REGION Network 6: InterLock
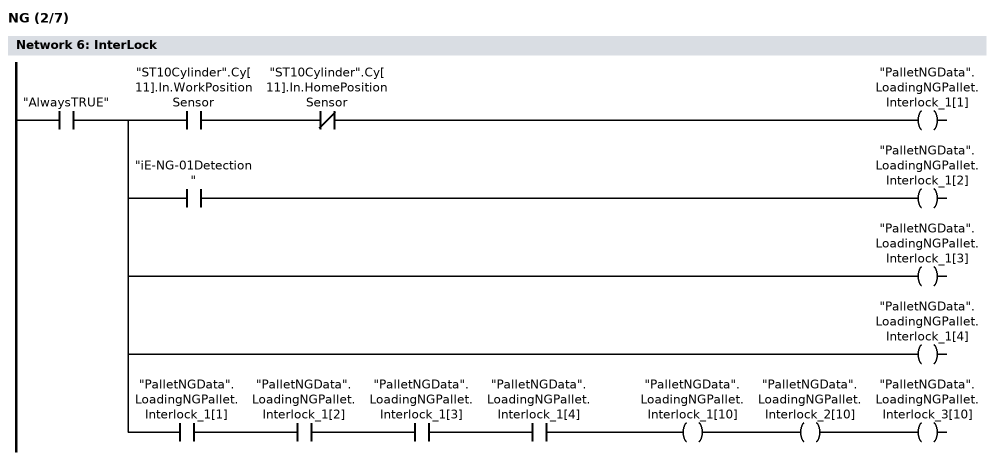
   RUNG wire#powerrail
      Contact( "AlwaysTRUE" )
      wire#w1
      Contact( "ST10Cylinder".Cy[11].In.WorkPositionSensor )
      I_Contact( "ST10Cylinder".Cy[11].In.HomePositionSensor )
      Coil( "PalletNGData".LoadingNGPallet.Interlock_1[1] )
   END_RUNG
   RUNG wire#w1
      Contact( "iE-NG-01Detection" )
      Coil( "PalletNGData".LoadingNGPallet.Interlock_1[2] )
   END_RUNG
   RUNG wire#w1
      Coil( "PalletNGData".LoadingNGPallet.Interlock_1[3] )
   END_RUNG
   RUNG wire#w1
      Coil( "PalletNGData".LoadingNGPallet.Interlock_1[4] )
   END_RUNG
   RUNG wire#w1
      Contact( "PalletNGData".LoadingNGPallet.Interlock_1[1] )
      Contact( "PalletNGData".LoadingNGPallet.Interlock_1[2] )
      Contact( "PalletNGData".LoadingNGPallet.Interlock_1[3] )
      Contact( "PalletNGData".LoadingNGPallet.Interlock_1[4] )
      Coil( "PalletNGData".LoadingNGPallet.Interlock_1[10] )
      Coil( "PalletNGData".LoadingNGPallet.Interlock_2[10] )
      Coil( "PalletNGData".LoadingNGPallet.Interlock_3[10] )
   END_RUNG
   // the same network as SCL:
   "PalletNGData".LoadingNGPallet.Interlock_1[1] := "AlwaysTRUE" AND "ST10Cylinder".Cy[11].In.WorkPositionSensor AND NOT "ST10Cylinder".Cy[11].In.HomePositionSensor;
   "PalletNGData".LoadingNGPallet.Interlock_1[2] := "AlwaysTRUE" AND "iE-NG-01Detection";
   "PalletNGData".LoadingNGPallet.Interlock_1[3] := "AlwaysTRUE";
   "PalletNGData".LoadingNGPallet.Interlock_1[4] := "AlwaysTRUE";
   #_w1 := "AlwaysTRUE" AND "PalletNGData".LoadingNGPallet.Interlock_1[1] AND "PalletNGData".LoadingNGPallet.Interlock_1[2] AND "PalletNGData".LoadingNGPallet.Interlock_1[3] AND "PalletNGData".LoadingNGPallet.Interlock_1[4];
   "PalletNGData".LoadingNGPallet.Interlock_1[10] := #_w1;
   "PalletNGData".LoadingNGPallet.Interlock_2[10] := #_w1;
   "PalletNGData".LoadingNGPallet.Interlock_3[10] := #_w1;
END_REGION

REGION Network 7: NG_Button
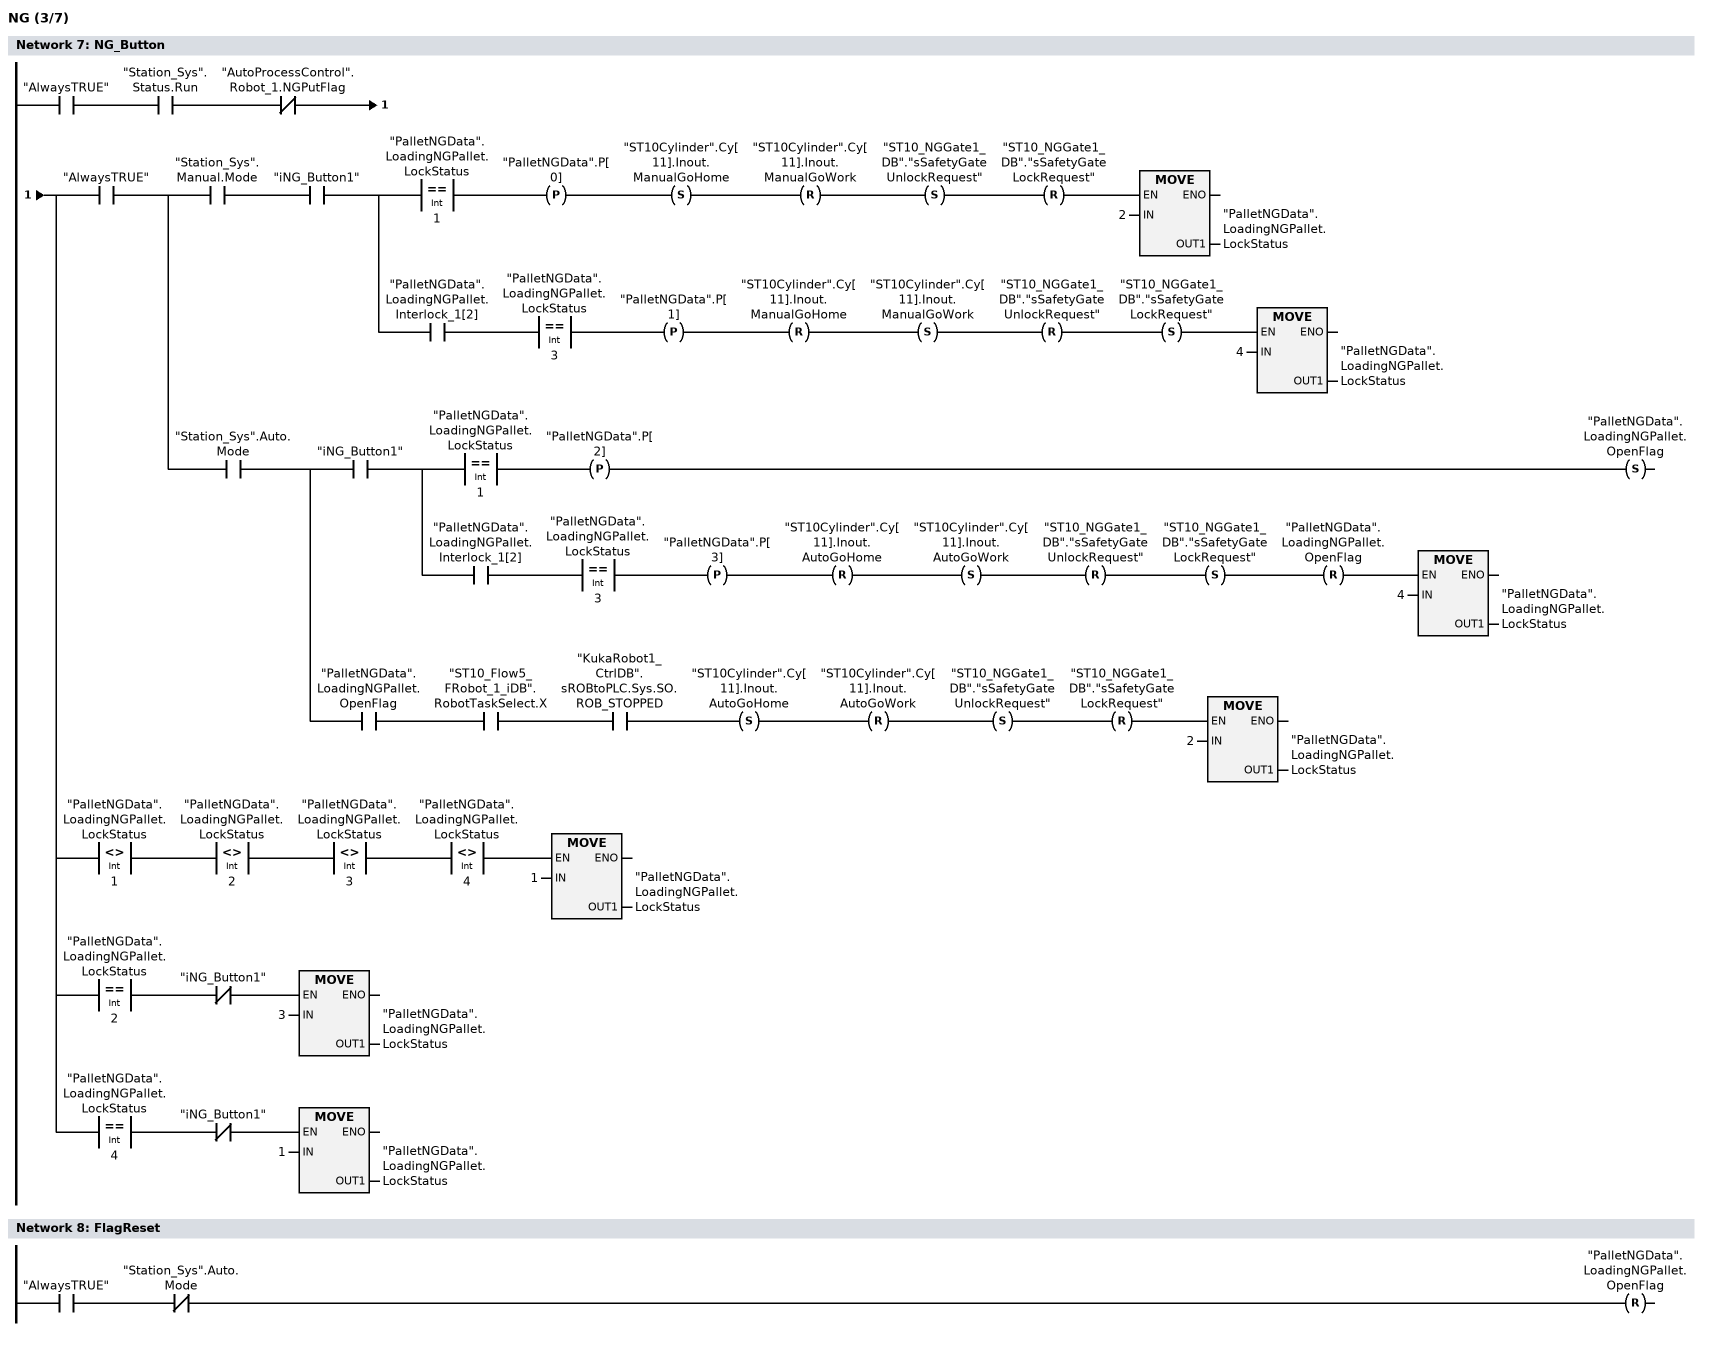
   RUNG wire#powerrail
      Contact( "AlwaysTRUE" )
      Contact( "Station_Sys".Status.Run )
      I_Contact( "AutoProcessControl".Robot_1.NGPutFlag )
      wire#w1
      Contact( "AlwaysTRUE" )
      wire#w2
      Contact( "Station_Sys".Manual.Mode )
      Contact( "iNG_Button1" )
      wire#w3
      { S7_Templates := "SrcType := Int" } EQ_Contact(in1 := "PalletNGData".LoadingNGPallet.LockStatus, in2 := 1)
      P_Trig( "PalletNGData".P[0] )
      S_Coil( "ST10Cylinder".Cy[11].Inout.ManualGoHome )
      R_Coil( "ST10Cylinder".Cy[11].Inout.ManualGoWork )
      S_Coil( "ST10_NGGate1_DB"."sSafetyGate UnlockRequest" )
      R_Coil( "ST10_NGGate1_DB"."sSafetyGate LockRequest" )
      Move(in := 2, out1 => "PalletNGData".LoadingNGPallet.LockStatus)
   END_RUNG
   RUNG wire#w3
      Contact( "PalletNGData".LoadingNGPallet.Interlock_1[2] )
      { S7_Templates := "SrcType := Int" } EQ_Contact(in1 := "PalletNGData".LoadingNGPallet.LockStatus, in2 := 3)
      P_Trig( "PalletNGData".P[1] )
      R_Coil( "ST10Cylinder".Cy[11].Inout.ManualGoHome )
      S_Coil( "ST10Cylinder".Cy[11].Inout.ManualGoWork )
      R_Coil( "ST10_NGGate1_DB"."sSafetyGate UnlockRequest" )
      S_Coil( "ST10_NGGate1_DB"."sSafetyGate LockRequest" )
      Move(in := 4, out1 => "PalletNGData".LoadingNGPallet.LockStatus)
   END_RUNG
   RUNG wire#w2
      Contact( "Station_Sys".Auto.Mode )
      wire#w4
      Contact( "iNG_Button1" )
      wire#w5
      { S7_Templates := "SrcType := Int" } EQ_Contact(in1 := "PalletNGData".LoadingNGPallet.LockStatus, in2 := 1)
      P_Trig( "PalletNGData".P[2] )
      S_Coil( "PalletNGData".LoadingNGPallet.OpenFlag )
   END_RUNG
   RUNG wire#w5
      Contact( "PalletNGData".LoadingNGPallet.Interlock_1[2] )
      { S7_Templates := "SrcType := Int" } EQ_Contact(in1 := "PalletNGData".LoadingNGPallet.LockStatus, in2 := 3)
      P_Trig( "PalletNGData".P[3] )
      R_Coil( "ST10Cylinder".Cy[11].Inout.AutoGoHome )
      S_Coil( "ST10Cylinder".Cy[11].Inout.AutoGoWork )
      R_Coil( "ST10_NGGate1_DB"."sSafetyGate UnlockRequest" )
      S_Coil( "ST10_NGGate1_DB"."sSafetyGate LockRequest" )
      R_Coil( "PalletNGData".LoadingNGPallet.OpenFlag )
      Move(in := 4, out1 => "PalletNGData".LoadingNGPallet.LockStatus)
   END_RUNG
   RUNG wire#w4
      Contact( "PalletNGData".LoadingNGPallet.OpenFlag )
      Contact( "ST10_Flow5_FRobot_1_iDB".RobotTaskSelect.X )
      Contact( "KukaRobot1_CtrlDB".sROBtoPLC.Sys.SO.ROB_STOPPED )
      S_Coil( "ST10Cylinder".Cy[11].Inout.AutoGoHome )
      R_Coil( "ST10Cylinder".Cy[11].Inout.AutoGoWork )
      S_Coil( "ST10_NGGate1_DB"."sSafetyGate UnlockRequest" )
      R_Coil( "ST10_NGGate1_DB"."sSafetyGate LockRequest" )
      Move(in := 2, out1 => "PalletNGData".LoadingNGPallet.LockStatus)
   END_RUNG
   RUNG wire#w1
      { S7_Templates := "SrcType := Int" } NE_Contact(in1 := "PalletNGData".LoadingNGPallet.LockStatus, in2 := 1)
      { S7_Templates := "SrcType := Int" } NE_Contact(in1 := "PalletNGData".LoadingNGPallet.LockStatus, in2 := 2)
      { S7_Templates := "SrcType := Int" } NE_Contact(in1 := "PalletNGData".LoadingNGPallet.LockStatus, in2 := 3)
      { S7_Templates := "SrcType := Int" } NE_Contact(in1 := "PalletNGData".LoadingNGPallet.LockStatus, in2 := 4)
      Move(in := 1, out1 => "PalletNGData".LoadingNGPallet.LockStatus)
   END_RUNG
   RUNG wire#w1
      { S7_Templates := "SrcType := Int" } EQ_Contact(in1 := "PalletNGData".LoadingNGPallet.LockStatus, in2 := 2)
      I_Contact( "iNG_Button1" )
      Move(in := 3, out1 => "PalletNGData".LoadingNGPallet.LockStatus)
   END_RUNG
   RUNG wire#w1
      { S7_Templates := "SrcType := Int" } EQ_Contact(in1 := "PalletNGData".LoadingNGPallet.LockStatus, in2 := 4)
      I_Contact( "iNG_Button1" )
      Move(in := 1, out1 => "PalletNGData".LoadingNGPallet.LockStatus)
   END_RUNG
   // the same network as SCL:
   #_w1 := "AlwaysTRUE" AND "Station_Sys".Status.Run AND NOT "AutoProcessControl".Robot_1.NGPutFlag;
   #_w2 := #_w1 AND "AlwaysTRUE";
   #_w3 := #_w2 AND "Station_Sys".Manual.Mode AND "iNG_Button1";
   #_w4 := #_w3 AND ("PalletNGData".LoadingNGPallet.LockStatus = 1);
   #_w5 := #_w4 AND NOT "PalletNGData".P[0];   // rising edge
   "PalletNGData".P[0] := #_w4;
   IF #_w5 THEN
       "ST10Cylinder".Cy[11].Inout.ManualGoHome := TRUE;
       "ST10Cylinder".Cy[11].Inout.ManualGoWork := FALSE;
       "ST10_NGGate1_DB"."sSafetyGate UnlockRequest" := TRUE;
       "ST10_NGGate1_DB"."sSafetyGate LockRequest" := FALSE;
       "PalletNGData".LoadingNGPallet.LockStatus := 2;
   END_IF;
   #_w6 := #_w3 AND "PalletNGData".LoadingNGPallet.Interlock_1[2] AND ("PalletNGData".LoadingNGPallet.LockStatus = 3);
   #_w7 := #_w6 AND NOT "PalletNGData".P[1];   // rising edge
   "PalletNGData".P[1] := #_w6;
   IF #_w7 THEN
       "ST10Cylinder".Cy[11].Inout.ManualGoHome := FALSE;
       "ST10Cylinder".Cy[11].Inout.ManualGoWork := TRUE;
       "ST10_NGGate1_DB"."sSafetyGate UnlockRequest" := FALSE;
       "ST10_NGGate1_DB"."sSafetyGate LockRequest" := TRUE;
       "PalletNGData".LoadingNGPallet.LockStatus := 4;
   END_IF;
   #_w8 := #_w2 AND "Station_Sys".Auto.Mode;
   #_w9 := #_w8 AND "iNG_Button1";
   #_w10 := #_w9 AND ("PalletNGData".LoadingNGPallet.LockStatus = 1);
   #_w11 := #_w10 AND NOT "PalletNGData".P[2];   // rising edge
   "PalletNGData".P[2] := #_w10;
   IF #_w11 THEN "PalletNGData".LoadingNGPallet.OpenFlag := TRUE; END_IF;
   #_w12 := #_w9 AND "PalletNGData".LoadingNGPallet.Interlock_1[2] AND ("PalletNGData".LoadingNGPallet.LockStatus = 3);
   #_w13 := #_w12 AND NOT "PalletNGData".P[3];   // rising edge
   "PalletNGData".P[3] := #_w12;
   IF #_w13 THEN
       "ST10Cylinder".Cy[11].Inout.AutoGoHome := FALSE;
       "ST10Cylinder".Cy[11].Inout.AutoGoWork := TRUE;
       "ST10_NGGate1_DB"."sSafetyGate UnlockRequest" := FALSE;
       "ST10_NGGate1_DB"."sSafetyGate LockRequest" := TRUE;
       "PalletNGData".LoadingNGPallet.OpenFlag := FALSE;
       "PalletNGData".LoadingNGPallet.LockStatus := 4;
   END_IF;
   IF #_w8 AND "PalletNGData".LoadingNGPallet.OpenFlag AND "ST10_Flow5_FRobot_1_iDB".RobotTaskSelect.X AND "KukaRobot1_CtrlDB".sROBtoPLC.Sys.SO.ROB_STOPPED THEN
       "ST10Cylinder".Cy[11].Inout.AutoGoHome := TRUE;
       "ST10Cylinder".Cy[11].Inout.AutoGoWork := FALSE;
       "ST10_NGGate1_DB"."sSafetyGate UnlockRequest" := TRUE;
       "ST10_NGGate1_DB"."sSafetyGate LockRequest" := FALSE;
       "PalletNGData".LoadingNGPallet.LockStatus := 2;
   END_IF;
   IF #_w1 AND ("PalletNGData".LoadingNGPallet.LockStatus <> 1) AND ("PalletNGData".LoadingNGPallet.LockStatus <> 2) AND ("PalletNGData".LoadingNGPallet.LockStatus <> 3) AND ("PalletNGData".LoadingNGPallet.LockStatus <> 4) THEN
       "PalletNGData".LoadingNGPallet.LockStatus := 1;
   END_IF;
   IF #_w1 AND ("PalletNGData".LoadingNGPallet.LockStatus = 2) AND NOT "iNG_Button1" THEN
       "PalletNGData".LoadingNGPallet.LockStatus := 3;
   END_IF;
   IF #_w1 AND ("PalletNGData".LoadingNGPallet.LockStatus = 4) AND NOT "iNG_Button1" THEN
       "PalletNGData".LoadingNGPallet.LockStatus := 1;
   END_IF;
END_REGION

REGION Network 8: FlagReset
   RUNG wire#powerrail
      Contact( "AlwaysTRUE" )
      I_Contact( "Station_Sys".Auto.Mode )
      R_Coil( "PalletNGData".LoadingNGPallet.OpenFlag )
   END_RUNG
   // the same network as SCL:
   IF "AlwaysTRUE" AND NOT "Station_Sys".Auto.Mode THEN
       "PalletNGData".LoadingNGPallet.OpenFlag := FALSE;
   END_IF;
END_REGION

REGION Network 9: NG Door
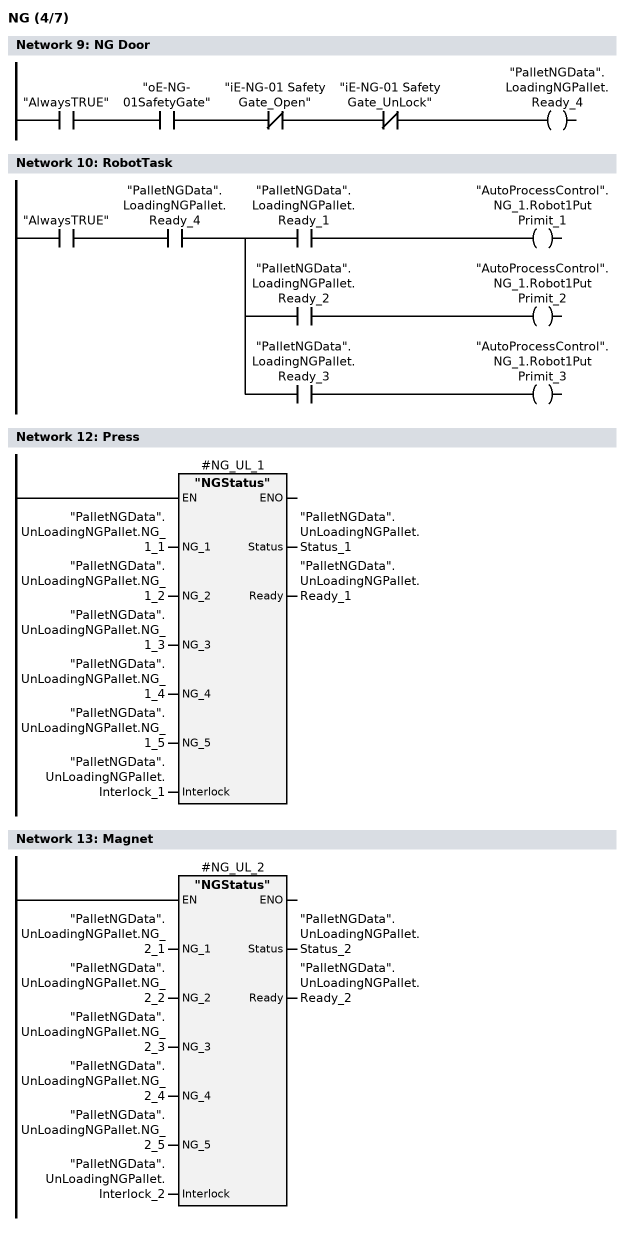
   RUNG wire#powerrail
      Contact( "AlwaysTRUE" )
      Contact( "oE-NG-01SafetyGate" )
      I_Contact( "iE-NG-01 Safety Gate_Open" )
      I_Contact( "iE-NG-01 Safety Gate_UnLock" )
      Coil( "PalletNGData".LoadingNGPallet.Ready_4 )
   END_RUNG
   // the same network as SCL:
   "PalletNGData".LoadingNGPallet.Ready_4 := "AlwaysTRUE" AND "oE-NG-01SafetyGate" AND NOT "iE-NG-01 Safety Gate_Open" AND NOT "iE-NG-01 Safety Gate_UnLock";
END_REGION

REGION Network 10: RobotTask
   RUNG wire#powerrail
      Contact( "AlwaysTRUE" )
      Contact( "PalletNGData".LoadingNGPallet.Ready_4 )
      wire#w1
      Contact( "PalletNGData".LoadingNGPallet.Ready_1 )
      Coil( "AutoProcessControl".NG_1.Robot1PutPrimit_1 )
   END_RUNG
   RUNG wire#w1
      Contact( "PalletNGData".LoadingNGPallet.Ready_2 )
      Coil( "AutoProcessControl".NG_1.Robot1PutPrimit_2 )
   END_RUNG
   RUNG wire#w1
      Contact( "PalletNGData".LoadingNGPallet.Ready_3 )
      Coil( "AutoProcessControl".NG_1.Robot1PutPrimit_3 )
   END_RUNG
   // the same network as SCL:
   #_w1 := "AlwaysTRUE" AND "PalletNGData".LoadingNGPallet.Ready_4;
   "AutoProcessControl".NG_1.Robot1PutPrimit_1 := #_w1 AND "PalletNGData".LoadingNGPallet.Ready_1;
   "AutoProcessControl".NG_1.Robot1PutPrimit_2 := #_w1 AND "PalletNGData".LoadingNGPallet.Ready_2;
   "AutoProcessControl".NG_1.Robot1PutPrimit_3 := #_w1 AND "PalletNGData".LoadingNGPallet.Ready_3;
END_REGION

REGION Network 11: --------------------------------------- UnLoad -------------------------------------------------------
END_REGION

REGION Network 12: Press
   RUNG wire#powerrail
      #NG_UL_1(NG_1 := "PalletNGData".UnLoadingNGPallet.NG_1_1, NG_2 := "PalletNGData".UnLoadingNGPallet.NG_1_2, NG_3 := "PalletNGData".UnLoadingNGPallet.NG_1_3, NG_4 := "PalletNGData".UnLoadingNGPallet.NG_1_4, NG_5 := "PalletNGData".UnLoadingNGPallet.NG_1_5, Interlock := "PalletNGData".UnLoadingNGPallet.Interlock_1, Status => "PalletNGData".UnLoadingNGPallet.Status_1, Ready => "PalletNGData".UnLoadingNGPallet.Ready_1)
   END_RUNG
   // the same network as SCL:
   #NG_UL_1(NG_1 := "PalletNGData".UnLoadingNGPallet.NG_1_1,   // "NGStatus"
            NG_2 := "PalletNGData".UnLoadingNGPallet.NG_1_2,
            NG_3 := "PalletNGData".UnLoadingNGPallet.NG_1_3,
            NG_4 := "PalletNGData".UnLoadingNGPallet.NG_1_4,
            NG_5 := "PalletNGData".UnLoadingNGPallet.NG_1_5,
            Interlock := "PalletNGData".UnLoadingNGPallet.Interlock_1,
            Status => "PalletNGData".UnLoadingNGPallet.Status_1,
            Ready => "PalletNGData".UnLoadingNGPallet.Ready_1);
END_REGION

REGION Network 13: Magnet
   RUNG wire#powerrail
      #NG_UL_2(NG_1 := "PalletNGData".UnLoadingNGPallet.NG_2_1, NG_2 := "PalletNGData".UnLoadingNGPallet.NG_2_2, NG_3 := "PalletNGData".UnLoadingNGPallet.NG_2_3, NG_4 := "PalletNGData".UnLoadingNGPallet.NG_2_4, NG_5 := "PalletNGData".UnLoadingNGPallet.NG_2_5, Interlock := "PalletNGData".UnLoadingNGPallet.Interlock_2, Status => "PalletNGData".UnLoadingNGPallet.Status_2, Ready => "PalletNGData".UnLoadingNGPallet.Ready_2)
   END_RUNG
   // the same network as SCL:
   #NG_UL_2(NG_1 := "PalletNGData".UnLoadingNGPallet.NG_2_1,   // "NGStatus"
            NG_2 := "PalletNGData".UnLoadingNGPallet.NG_2_2,
            NG_3 := "PalletNGData".UnLoadingNGPallet.NG_2_3,
            NG_4 := "PalletNGData".UnLoadingNGPallet.NG_2_4,
            NG_5 := "PalletNGData".UnLoadingNGPallet.NG_2_5,
            Interlock := "PalletNGData".UnLoadingNGPallet.Interlock_2,
            Status => "PalletNGData".UnLoadingNGPallet.Status_2,
            Ready => "PalletNGData".UnLoadingNGPallet.Ready_2);
END_REGION

REGION Network 14: Ring
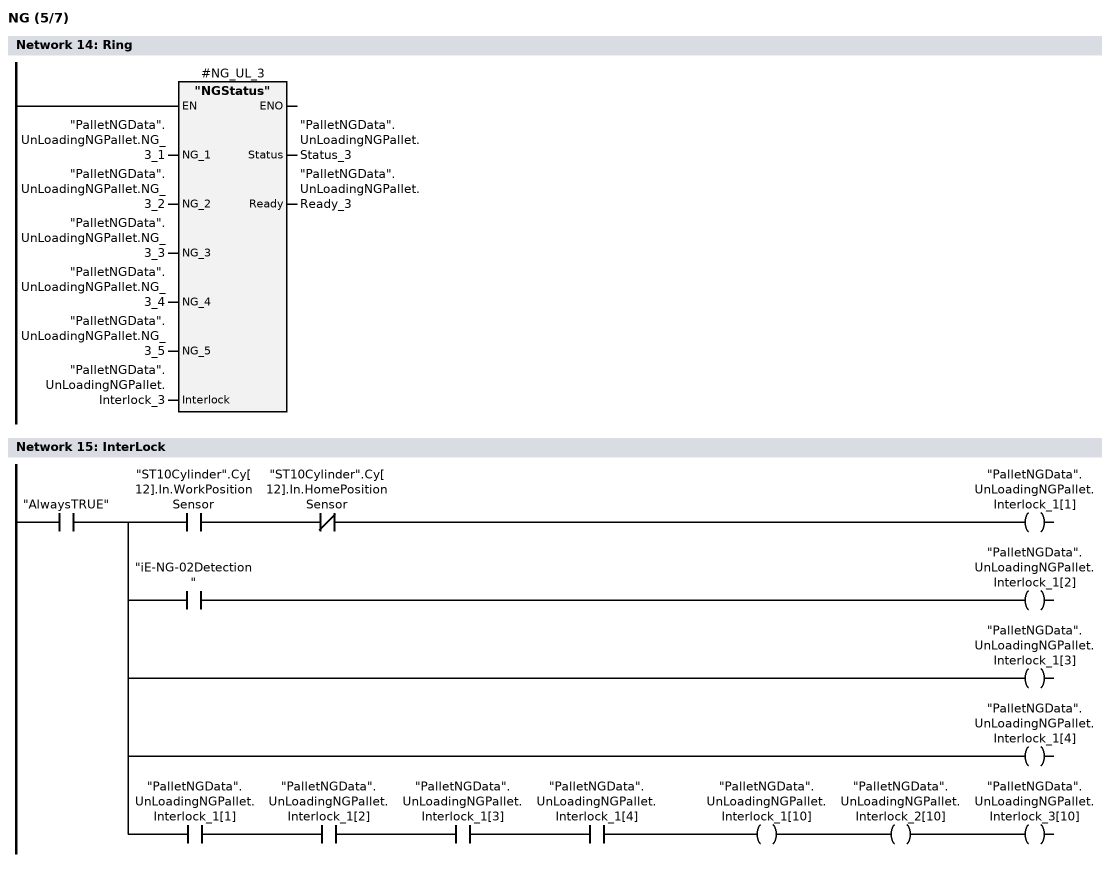
   RUNG wire#powerrail
      #NG_UL_3(NG_1 := "PalletNGData".UnLoadingNGPallet.NG_3_1, NG_2 := "PalletNGData".UnLoadingNGPallet.NG_3_2, NG_3 := "PalletNGData".UnLoadingNGPallet.NG_3_3, NG_4 := "PalletNGData".UnLoadingNGPallet.NG_3_4, NG_5 := "PalletNGData".UnLoadingNGPallet.NG_3_5, Interlock := "PalletNGData".UnLoadingNGPallet.Interlock_3, Status => "PalletNGData".UnLoadingNGPallet.Status_3, Ready => "PalletNGData".UnLoadingNGPallet.Ready_3)
   END_RUNG
   // the same network as SCL:
   #NG_UL_3(NG_1 := "PalletNGData".UnLoadingNGPallet.NG_3_1,   // "NGStatus"
            NG_2 := "PalletNGData".UnLoadingNGPallet.NG_3_2,
            NG_3 := "PalletNGData".UnLoadingNGPallet.NG_3_3,
            NG_4 := "PalletNGData".UnLoadingNGPallet.NG_3_4,
            NG_5 := "PalletNGData".UnLoadingNGPallet.NG_3_5,
            Interlock := "PalletNGData".UnLoadingNGPallet.Interlock_3,
            Status => "PalletNGData".UnLoadingNGPallet.Status_3,
            Ready => "PalletNGData".UnLoadingNGPallet.Ready_3);
END_REGION

REGION Network 15: InterLock
   RUNG wire#powerrail
      Contact( "AlwaysTRUE" )
      wire#w1
      Contact( "ST10Cylinder".Cy[12].In.WorkPositionSensor )
      I_Contact( "ST10Cylinder".Cy[12].In.HomePositionSensor )
      Coil( "PalletNGData".UnLoadingNGPallet.Interlock_1[1] )
   END_RUNG
   RUNG wire#w1
      Contact( "iE-NG-02Detection" )
      Coil( "PalletNGData".UnLoadingNGPallet.Interlock_1[2] )
   END_RUNG
   RUNG wire#w1
      Coil( "PalletNGData".UnLoadingNGPallet.Interlock_1[3] )
   END_RUNG
   RUNG wire#w1
      Coil( "PalletNGData".UnLoadingNGPallet.Interlock_1[4] )
   END_RUNG
   RUNG wire#w1
      Contact( "PalletNGData".UnLoadingNGPallet.Interlock_1[1] )
      Contact( "PalletNGData".UnLoadingNGPallet.Interlock_1[2] )
      Contact( "PalletNGData".UnLoadingNGPallet.Interlock_1[3] )
      Contact( "PalletNGData".UnLoadingNGPallet.Interlock_1[4] )
      Coil( "PalletNGData".UnLoadingNGPallet.Interlock_1[10] )
      Coil( "PalletNGData".UnLoadingNGPallet.Interlock_2[10] )
      Coil( "PalletNGData".UnLoadingNGPallet.Interlock_3[10] )
   END_RUNG
   // the same network as SCL:
   "PalletNGData".UnLoadingNGPallet.Interlock_1[1] := "AlwaysTRUE" AND "ST10Cylinder".Cy[12].In.WorkPositionSensor AND NOT "ST10Cylinder".Cy[12].In.HomePositionSensor;
   "PalletNGData".UnLoadingNGPallet.Interlock_1[2] := "AlwaysTRUE" AND "iE-NG-02Detection";
   "PalletNGData".UnLoadingNGPallet.Interlock_1[3] := "AlwaysTRUE";
   "PalletNGData".UnLoadingNGPallet.Interlock_1[4] := "AlwaysTRUE";
   #_w1 := "AlwaysTRUE" AND "PalletNGData".UnLoadingNGPallet.Interlock_1[1] AND "PalletNGData".UnLoadingNGPallet.Interlock_1[2] AND "PalletNGData".UnLoadingNGPallet.Interlock_1[3] AND "PalletNGData".UnLoadingNGPallet.Interlock_1[4];
   "PalletNGData".UnLoadingNGPallet.Interlock_1[10] := #_w1;
   "PalletNGData".UnLoadingNGPallet.Interlock_2[10] := #_w1;
   "PalletNGData".UnLoadingNGPallet.Interlock_3[10] := #_w1;
END_REGION

REGION Network 16: NG_Button
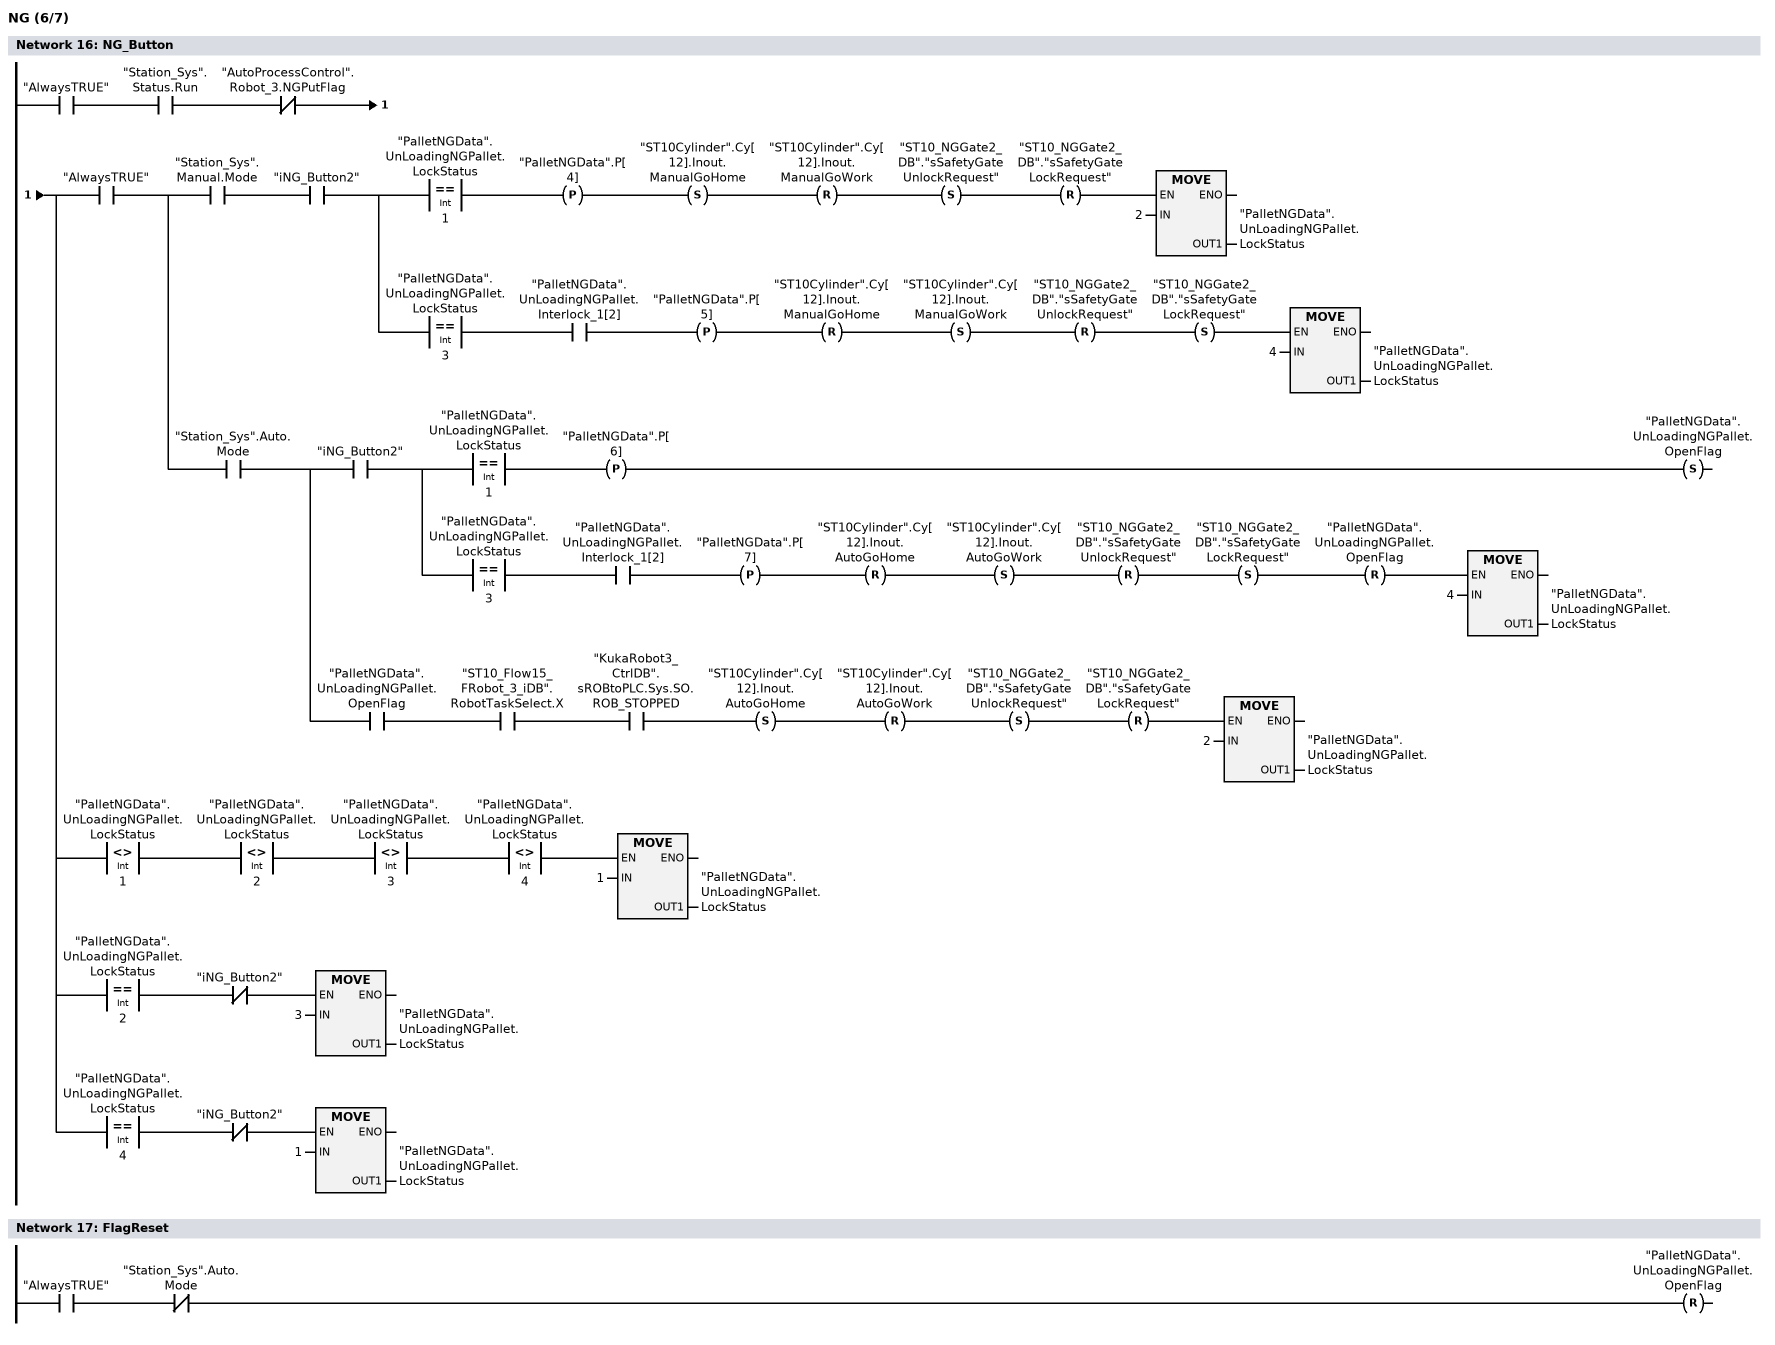
   RUNG wire#powerrail
      Contact( "AlwaysTRUE" )
      Contact( "Station_Sys".Status.Run )
      I_Contact( "AutoProcessControl".Robot_3.NGPutFlag )
      wire#w1
      Contact( "AlwaysTRUE" )
      wire#w2
      Contact( "Station_Sys".Manual.Mode )
      Contact( "iNG_Button2" )
      wire#w3
      { S7_Templates := "SrcType := Int" } EQ_Contact(in1 := "PalletNGData".UnLoadingNGPallet.LockStatus, in2 := 1)
      P_Trig( "PalletNGData".P[4] )
      S_Coil( "ST10Cylinder".Cy[12].Inout.ManualGoHome )
      R_Coil( "ST10Cylinder".Cy[12].Inout.ManualGoWork )
      S_Coil( "ST10_NGGate2_DB"."sSafetyGate UnlockRequest" )
      R_Coil( "ST10_NGGate2_DB"."sSafetyGate LockRequest" )
      Move(in := 2, out1 => "PalletNGData".UnLoadingNGPallet.LockStatus)
   END_RUNG
   RUNG wire#w3
      { S7_Templates := "SrcType := Int" } EQ_Contact(in1 := "PalletNGData".UnLoadingNGPallet.LockStatus, in2 := 3)
      Contact( "PalletNGData".UnLoadingNGPallet.Interlock_1[2] )
      P_Trig( "PalletNGData".P[5] )
      R_Coil( "ST10Cylinder".Cy[12].Inout.ManualGoHome )
      S_Coil( "ST10Cylinder".Cy[12].Inout.ManualGoWork )
      R_Coil( "ST10_NGGate2_DB"."sSafetyGate UnlockRequest" )
      S_Coil( "ST10_NGGate2_DB"."sSafetyGate LockRequest" )
      Move(in := 4, out1 => "PalletNGData".UnLoadingNGPallet.LockStatus)
   END_RUNG
   RUNG wire#w2
      Contact( "Station_Sys".Auto.Mode )
      wire#w4
      Contact( "iNG_Button2" )
      wire#w5
      { S7_Templates := "SrcType := Int" } EQ_Contact(in1 := "PalletNGData".UnLoadingNGPallet.LockStatus, in2 := 1)
      P_Trig( "PalletNGData".P[6] )
      S_Coil( "PalletNGData".UnLoadingNGPallet.OpenFlag )
   END_RUNG
   RUNG wire#w5
      { S7_Templates := "SrcType := Int" } EQ_Contact(in1 := "PalletNGData".UnLoadingNGPallet.LockStatus, in2 := 3)
      Contact( "PalletNGData".UnLoadingNGPallet.Interlock_1[2] )
      P_Trig( "PalletNGData".P[7] )
      R_Coil( "ST10Cylinder".Cy[12].Inout.AutoGoHome )
      S_Coil( "ST10Cylinder".Cy[12].Inout.AutoGoWork )
      R_Coil( "ST10_NGGate2_DB"."sSafetyGate UnlockRequest" )
      S_Coil( "ST10_NGGate2_DB"."sSafetyGate LockRequest" )
      R_Coil( "PalletNGData".UnLoadingNGPallet.OpenFlag )
      Move(in := 4, out1 => "PalletNGData".UnLoadingNGPallet.LockStatus)
   END_RUNG
   RUNG wire#w4
      Contact( "PalletNGData".UnLoadingNGPallet.OpenFlag )
      Contact( "ST10_Flow15_FRobot_3_iDB".RobotTaskSelect.X )
      Contact( "KukaRobot3_CtrlDB".sROBtoPLC.Sys.SO.ROB_STOPPED )
      S_Coil( "ST10Cylinder".Cy[12].Inout.AutoGoHome )
      R_Coil( "ST10Cylinder".Cy[12].Inout.AutoGoWork )
      S_Coil( "ST10_NGGate2_DB"."sSafetyGate UnlockRequest" )
      R_Coil( "ST10_NGGate2_DB"."sSafetyGate LockRequest" )
      Move(in := 2, out1 => "PalletNGData".UnLoadingNGPallet.LockStatus)
   END_RUNG
   RUNG wire#w1
      { S7_Templates := "SrcType := Int" } NE_Contact(in1 := "PalletNGData".UnLoadingNGPallet.LockStatus, in2 := 1)
      { S7_Templates := "SrcType := Int" } NE_Contact(in1 := "PalletNGData".UnLoadingNGPallet.LockStatus, in2 := 2)
      { S7_Templates := "SrcType := Int" } NE_Contact(in1 := "PalletNGData".UnLoadingNGPallet.LockStatus, in2 := 3)
      { S7_Templates := "SrcType := Int" } NE_Contact(in1 := "PalletNGData".UnLoadingNGPallet.LockStatus, in2 := 4)
      Move(in := 1, out1 => "PalletNGData".UnLoadingNGPallet.LockStatus)
   END_RUNG
   RUNG wire#w1
      { S7_Templates := "SrcType := Int" } EQ_Contact(in1 := "PalletNGData".UnLoadingNGPallet.LockStatus, in2 := 2)
      I_Contact( "iNG_Button2" )
      Move(in := 3, out1 => "PalletNGData".UnLoadingNGPallet.LockStatus)
   END_RUNG
   RUNG wire#w1
      { S7_Templates := "SrcType := Int" } EQ_Contact(in1 := "PalletNGData".UnLoadingNGPallet.LockStatus, in2 := 4)
      I_Contact( "iNG_Button2" )
      Move(in := 1, out1 => "PalletNGData".UnLoadingNGPallet.LockStatus)
   END_RUNG
   // the same network as SCL:
   #_w1 := "AlwaysTRUE" AND "Station_Sys".Status.Run AND NOT "AutoProcessControl".Robot_3.NGPutFlag;
   #_w2 := #_w1 AND "AlwaysTRUE";
   #_w3 := #_w2 AND "Station_Sys".Manual.Mode AND "iNG_Button2";
   #_w4 := #_w3 AND ("PalletNGData".UnLoadingNGPallet.LockStatus = 1);
   #_w5 := #_w4 AND NOT "PalletNGData".P[4];   // rising edge
   "PalletNGData".P[4] := #_w4;
   IF #_w5 THEN
       "ST10Cylinder".Cy[12].Inout.ManualGoHome := TRUE;
       "ST10Cylinder".Cy[12].Inout.ManualGoWork := FALSE;
       "ST10_NGGate2_DB"."sSafetyGate UnlockRequest" := TRUE;
       "ST10_NGGate2_DB"."sSafetyGate LockRequest" := FALSE;
       "PalletNGData".UnLoadingNGPallet.LockStatus := 2;
   END_IF;
   #_w6 := #_w3 AND ("PalletNGData".UnLoadingNGPallet.LockStatus = 3) AND "PalletNGData".UnLoadingNGPallet.Interlock_1[2];
   #_w7 := #_w6 AND NOT "PalletNGData".P[5];   // rising edge
   "PalletNGData".P[5] := #_w6;
   IF #_w7 THEN
       "ST10Cylinder".Cy[12].Inout.ManualGoHome := FALSE;
       "ST10Cylinder".Cy[12].Inout.ManualGoWork := TRUE;
       "ST10_NGGate2_DB"."sSafetyGate UnlockRequest" := FALSE;
       "ST10_NGGate2_DB"."sSafetyGate LockRequest" := TRUE;
       "PalletNGData".UnLoadingNGPallet.LockStatus := 4;
   END_IF;
   #_w8 := #_w2 AND "Station_Sys".Auto.Mode;
   #_w9 := #_w8 AND "iNG_Button2";
   #_w10 := #_w9 AND ("PalletNGData".UnLoadingNGPallet.LockStatus = 1);
   #_w11 := #_w10 AND NOT "PalletNGData".P[6];   // rising edge
   "PalletNGData".P[6] := #_w10;
   IF #_w11 THEN "PalletNGData".UnLoadingNGPallet.OpenFlag := TRUE; END_IF;
   #_w12 := #_w9 AND ("PalletNGData".UnLoadingNGPallet.LockStatus = 3) AND "PalletNGData".UnLoadingNGPallet.Interlock_1[2];
   #_w13 := #_w12 AND NOT "PalletNGData".P[7];   // rising edge
   "PalletNGData".P[7] := #_w12;
   IF #_w13 THEN
       "ST10Cylinder".Cy[12].Inout.AutoGoHome := FALSE;
       "ST10Cylinder".Cy[12].Inout.AutoGoWork := TRUE;
       "ST10_NGGate2_DB"."sSafetyGate UnlockRequest" := FALSE;
       "ST10_NGGate2_DB"."sSafetyGate LockRequest" := TRUE;
       "PalletNGData".UnLoadingNGPallet.OpenFlag := FALSE;
       "PalletNGData".UnLoadingNGPallet.LockStatus := 4;
   END_IF;
   IF #_w8 AND "PalletNGData".UnLoadingNGPallet.OpenFlag AND "ST10_Flow15_FRobot_3_iDB".RobotTaskSelect.X AND "KukaRobot3_CtrlDB".sROBtoPLC.Sys.SO.ROB_STOPPED THEN
       "ST10Cylinder".Cy[12].Inout.AutoGoHome := TRUE;
       "ST10Cylinder".Cy[12].Inout.AutoGoWork := FALSE;
       "ST10_NGGate2_DB"."sSafetyGate UnlockRequest" := TRUE;
       "ST10_NGGate2_DB"."sSafetyGate LockRequest" := FALSE;
       "PalletNGData".UnLoadingNGPallet.LockStatus := 2;
   END_IF;
   IF #_w1 AND ("PalletNGData".UnLoadingNGPallet.LockStatus <> 1) AND ("PalletNGData".UnLoadingNGPallet.LockStatus <> 2) AND ("PalletNGData".UnLoadingNGPallet.LockStatus <> 3) AND ("PalletNGData".UnLoadingNGPallet.LockStatus <> 4) THEN
       "PalletNGData".UnLoadingNGPallet.LockStatus := 1;
   END_IF;
   IF #_w1 AND ("PalletNGData".UnLoadingNGPallet.LockStatus = 2) AND NOT "iNG_Button2" THEN
       "PalletNGData".UnLoadingNGPallet.LockStatus := 3;
   END_IF;
   IF #_w1 AND ("PalletNGData".UnLoadingNGPallet.LockStatus = 4) AND NOT "iNG_Button2" THEN
       "PalletNGData".UnLoadingNGPallet.LockStatus := 1;
   END_IF;
END_REGION

REGION Network 17: FlagReset
   RUNG wire#powerrail
      Contact( "AlwaysTRUE" )
      I_Contact( "Station_Sys".Auto.Mode )
      R_Coil( "PalletNGData".UnLoadingNGPallet.OpenFlag )
   END_RUNG
   // the same network as SCL:
   IF "AlwaysTRUE" AND NOT "Station_Sys".Auto.Mode THEN
       "PalletNGData".UnLoadingNGPallet.OpenFlag := FALSE;
   END_IF;
END_REGION

REGION Network 18: NG Door
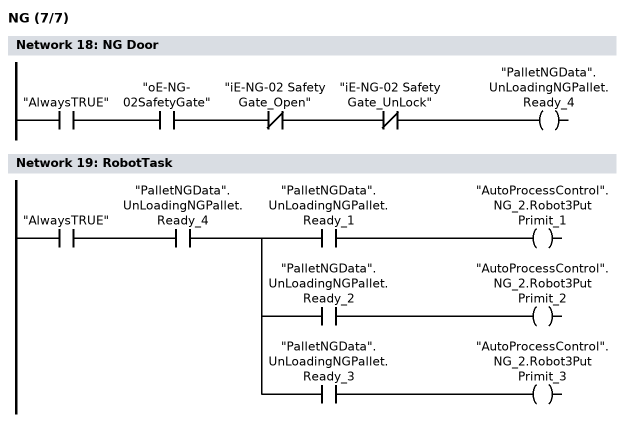
   RUNG wire#powerrail
      Contact( "AlwaysTRUE" )
      Contact( "oE-NG-02SafetyGate" )
      I_Contact( "iE-NG-02 Safety Gate_Open" )
      I_Contact( "iE-NG-02 Safety Gate_UnLock" )
      Coil( "PalletNGData".UnLoadingNGPallet.Ready_4 )
   END_RUNG
   // the same network as SCL:
   "PalletNGData".UnLoadingNGPallet.Ready_4 := "AlwaysTRUE" AND "oE-NG-02SafetyGate" AND NOT "iE-NG-02 Safety Gate_Open" AND NOT "iE-NG-02 Safety Gate_UnLock";
END_REGION

REGION Network 19: RobotTask
   RUNG wire#powerrail
      Contact( "AlwaysTRUE" )
      Contact( "PalletNGData".UnLoadingNGPallet.Ready_4 )
      wire#w1
      Contact( "PalletNGData".UnLoadingNGPallet.Ready_1 )
      Coil( "AutoProcessControl".NG_2.Robot3PutPrimit_1 )
   END_RUNG
   RUNG wire#w1
      Contact( "PalletNGData".UnLoadingNGPallet.Ready_2 )
      Coil( "AutoProcessControl".NG_2.Robot3PutPrimit_2 )
   END_RUNG
   RUNG wire#w1
      Contact( "PalletNGData".UnLoadingNGPallet.Ready_3 )
      Coil( "AutoProcessControl".NG_2.Robot3PutPrimit_3 )
   END_RUNG
   // the same network as SCL:
   #_w1 := "AlwaysTRUE" AND "PalletNGData".UnLoadingNGPallet.Ready_4;
   "AutoProcessControl".NG_2.Robot3PutPrimit_1 := #_w1 AND "PalletNGData".UnLoadingNGPallet.Ready_1;
   "AutoProcessControl".NG_2.Robot3PutPrimit_2 := #_w1 AND "PalletNGData".UnLoadingNGPallet.Ready_2;
   "AutoProcessControl".NG_2.Robot3PutPrimit_3 := #_w1 AND "PalletNGData".UnLoadingNGPallet.Ready_3;
END_REGION
END_FUNCTION_BLOCK

FUNCTION_BLOCK "NGStatus"   // FB2900, LAD
{ S7_Optimized_Access := 'TRUE' }
VERSION : 0.1
// stored: AutoNumber false, IsIECCheckEnabled false, IsRetainMemResEnabled false, MemoryReserve 100, SetENOAutomatically false, UDAEnableTagReadback false
   VAR_INPUT
      NG_1 : Bool;
      NG_2 : Bool;
      NG_3 : Bool;
      NG_4 : Bool;
      NG_5 : Bool;
   END_VAR
   VAR_OUTPUT
      Status : Int;
      Ready : Bool;
   END_VAR
   VAR_IN_OUT
      Interlock : Array[1..10] of Bool;
   END_VAR
   VAR
      AlwaysOn : Bool;
      NG_Delay : Array[1..10] of TON_TIME;
      NG_DelayTime { S7_SetPoint := 'True'} : Array[1..10] of DInt;
   END_VAR
   // NG_DelayTime[1..10] := 1000;
BEGIN

REGION Network 1: #AlwaysOn
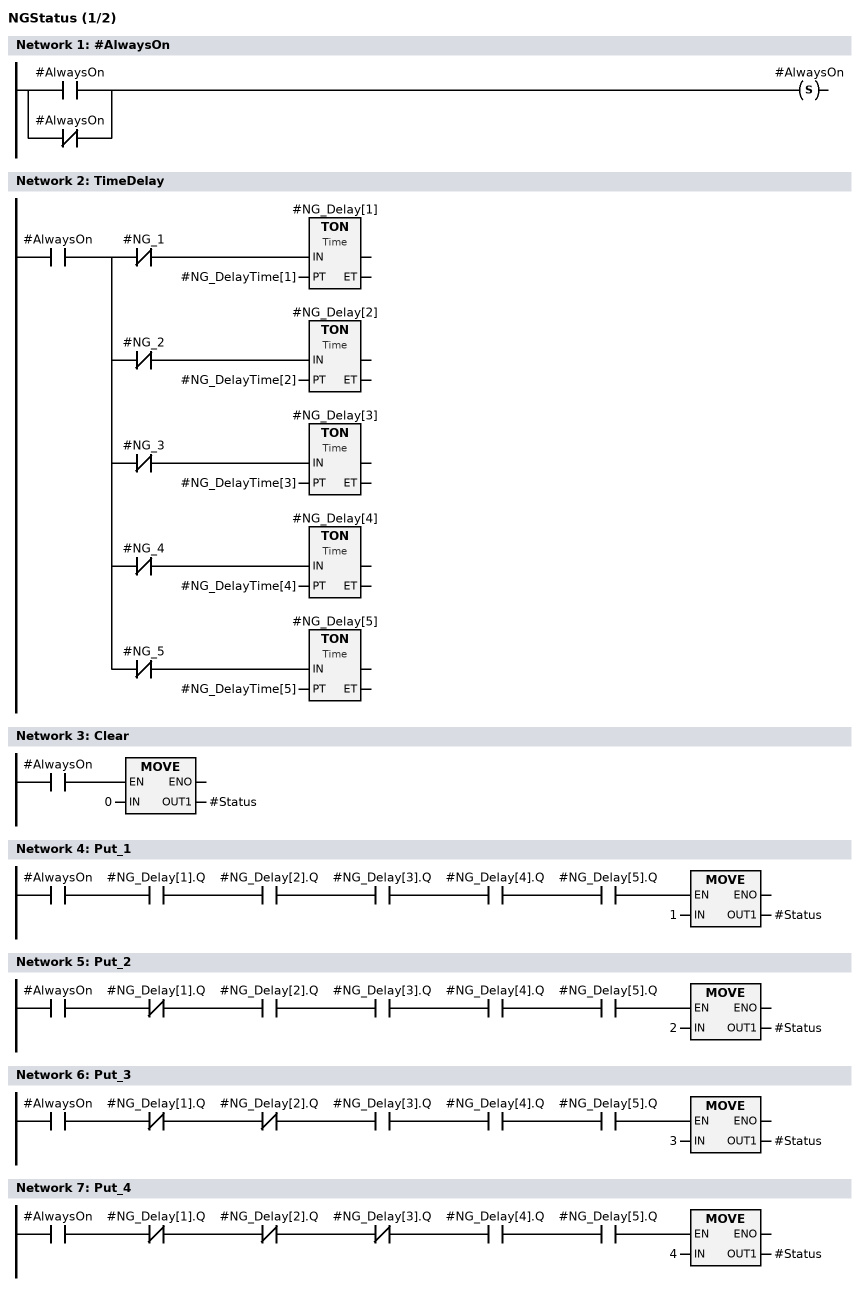
   RUNG wire#powerrail
      Contact( #AlwaysOn )
      wire#w1
      S_Coil( #AlwaysOn )
   END_RUNG
   RUNG wire#powerrail
      I_Contact( #AlwaysOn )
   END_RUNG wire#w1
   // the same network as SCL:
   IF #AlwaysOn OR NOT #AlwaysOn THEN #AlwaysOn := TRUE; END_IF;
END_REGION

REGION Network 2: TimeDelay
   RUNG wire#powerrail
      Contact( #AlwaysOn )
      wire#w1
      I_Contact( #NG_1 )
      { S7_Templates := "time_type := Time" } #NG_Delay[1].TON(pt := #NG_DelayTime[1], et =>)
   END_RUNG
   RUNG wire#w1
      I_Contact( #NG_2 )
      { S7_Templates := "time_type := Time" } #NG_Delay[2].TON(pt := #NG_DelayTime[2], et =>)
   END_RUNG
   RUNG wire#w1
      I_Contact( #NG_3 )
      { S7_Templates := "time_type := Time" } #NG_Delay[3].TON(pt := #NG_DelayTime[3], et =>)
   END_RUNG
   RUNG wire#w1
      I_Contact( #NG_4 )
      { S7_Templates := "time_type := Time" } #NG_Delay[4].TON(pt := #NG_DelayTime[4], et =>)
   END_RUNG
   RUNG wire#w1
      I_Contact( #NG_5 )
      { S7_Templates := "time_type := Time" } #NG_Delay[5].TON(pt := #NG_DelayTime[5], et =>)
   END_RUNG
   // the same network as SCL:
   #NG_Delay[1].TON(IN := #AlwaysOn AND NOT #NG_1, PT := #NG_DelayTime[1]);
   #NG_Delay[2].TON(IN := #AlwaysOn AND NOT #NG_2, PT := #NG_DelayTime[2]);
   #NG_Delay[3].TON(IN := #AlwaysOn AND NOT #NG_3, PT := #NG_DelayTime[3]);
   #NG_Delay[4].TON(IN := #AlwaysOn AND NOT #NG_4, PT := #NG_DelayTime[4]);
   #NG_Delay[5].TON(IN := #AlwaysOn AND NOT #NG_5, PT := #NG_DelayTime[5]);
END_REGION

REGION Network 3: Clear
   RUNG wire#powerrail
      Contact( #AlwaysOn )
      Move(in := 0, out1 => #Status)
   END_RUNG
   // the same network as SCL:
   IF #AlwaysOn THEN #Status := 0; END_IF;
END_REGION

REGION Network 4: Put_1
   RUNG wire#powerrail
      Contact( #AlwaysOn )
      Contact( #NG_Delay[1].Q )
      Contact( #NG_Delay[2].Q )
      Contact( #NG_Delay[3].Q )
      Contact( #NG_Delay[4].Q )
      Contact( #NG_Delay[5].Q )
      Move(in := 1, out1 => #Status)
   END_RUNG
   // the same network as SCL:
   IF #AlwaysOn AND #NG_Delay[1].Q AND #NG_Delay[2].Q AND #NG_Delay[3].Q AND #NG_Delay[4].Q AND #NG_Delay[5].Q THEN
       #Status := 1;
   END_IF;
END_REGION

REGION Network 5: Put_2
   RUNG wire#powerrail
      Contact( #AlwaysOn )
      I_Contact( #NG_Delay[1].Q )
      Contact( #NG_Delay[2].Q )
      Contact( #NG_Delay[3].Q )
      Contact( #NG_Delay[4].Q )
      Contact( #NG_Delay[5].Q )
      Move(in := 2, out1 => #Status)
   END_RUNG
   // the same network as SCL:
   IF #AlwaysOn AND NOT #NG_Delay[1].Q AND #NG_Delay[2].Q AND #NG_Delay[3].Q AND #NG_Delay[4].Q AND #NG_Delay[5].Q THEN
       #Status := 2;
   END_IF;
END_REGION

REGION Network 6: Put_3
   RUNG wire#powerrail
      Contact( #AlwaysOn )
      I_Contact( #NG_Delay[1].Q )
      I_Contact( #NG_Delay[2].Q )
      Contact( #NG_Delay[3].Q )
      Contact( #NG_Delay[4].Q )
      Contact( #NG_Delay[5].Q )
      Move(in := 3, out1 => #Status)
   END_RUNG
   // the same network as SCL:
   IF #AlwaysOn AND NOT #NG_Delay[1].Q AND NOT #NG_Delay[2].Q AND #NG_Delay[3].Q AND #NG_Delay[4].Q AND #NG_Delay[5].Q THEN
       #Status := 3;
   END_IF;
END_REGION

REGION Network 7: Put_4
   RUNG wire#powerrail
      Contact( #AlwaysOn )
      I_Contact( #NG_Delay[1].Q )
      I_Contact( #NG_Delay[2].Q )
      I_Contact( #NG_Delay[3].Q )
      Contact( #NG_Delay[4].Q )
      Contact( #NG_Delay[5].Q )
      Move(in := 4, out1 => #Status)
   END_RUNG
   // the same network as SCL:
   IF #AlwaysOn AND NOT #NG_Delay[1].Q AND NOT #NG_Delay[2].Q AND NOT #NG_Delay[3].Q AND #NG_Delay[4].Q AND #NG_Delay[5].Q THEN
       #Status := 4;
   END_IF;
END_REGION

REGION Network 8: Put_5
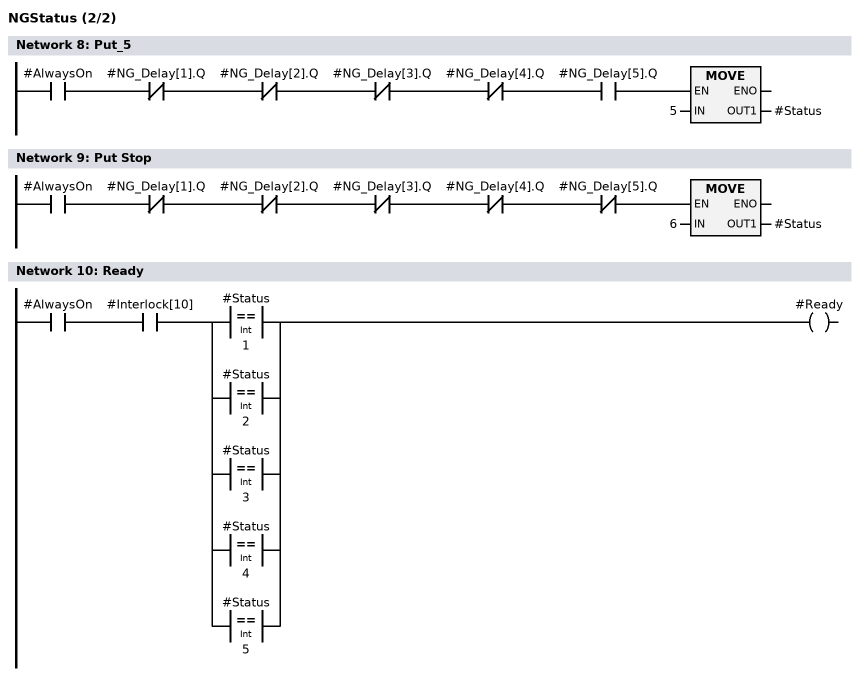
   RUNG wire#powerrail
      Contact( #AlwaysOn )
      I_Contact( #NG_Delay[1].Q )
      I_Contact( #NG_Delay[2].Q )
      I_Contact( #NG_Delay[3].Q )
      I_Contact( #NG_Delay[4].Q )
      Contact( #NG_Delay[5].Q )
      Move(in := 5, out1 => #Status)
   END_RUNG
   // the same network as SCL:
   IF #AlwaysOn AND NOT #NG_Delay[1].Q AND NOT #NG_Delay[2].Q AND NOT #NG_Delay[3].Q AND NOT #NG_Delay[4].Q AND #NG_Delay[5].Q THEN
       #Status := 5;
   END_IF;
END_REGION

REGION Network 9: Put Stop
   RUNG wire#powerrail
      Contact( #AlwaysOn )
      I_Contact( #NG_Delay[1].Q )
      I_Contact( #NG_Delay[2].Q )
      I_Contact( #NG_Delay[3].Q )
      I_Contact( #NG_Delay[4].Q )
      I_Contact( #NG_Delay[5].Q )
      Move(in := 6, out1 => #Status)
   END_RUNG
   // the same network as SCL:
   IF #AlwaysOn AND NOT #NG_Delay[1].Q AND NOT #NG_Delay[2].Q AND NOT #NG_Delay[3].Q AND NOT #NG_Delay[4].Q AND NOT #NG_Delay[5].Q THEN
       #Status := 6;
   END_IF;
END_REGION

REGION Network 10: Ready
   RUNG wire#powerrail
      Contact( #AlwaysOn )
      Contact( #Interlock[10] )
      wire#w1
      { S7_Templates := "SrcType := Int" } EQ_Contact(in1 := #Status, in2 := 1)
      wire#w2
      Coil( #Ready )
   END_RUNG
   RUNG wire#w1
      { S7_Templates := "SrcType := Int" } EQ_Contact(in1 := #Status, in2 := 2)
   END_RUNG wire#w2
   RUNG wire#w1
      { S7_Templates := "SrcType := Int" } EQ_Contact(in1 := #Status, in2 := 3)
   END_RUNG wire#w2
   RUNG wire#w1
      { S7_Templates := "SrcType := Int" } EQ_Contact(in1 := #Status, in2 := 4)
   END_RUNG wire#w2
   RUNG wire#w1
      { S7_Templates := "SrcType := Int" } EQ_Contact(in1 := #Status, in2 := 5)
   END_RUNG wire#w2
   // the same network as SCL:
   #Ready := #AlwaysOn AND #Interlock[10] AND ((#Status = 1) OR (#Status = 2) OR (#Status = 3) OR (#Status = 4) OR (#Status = 5));
END_REGION
END_FUNCTION_BLOCK

FUNCTION_BLOCK "FB_Next"   // FB42, SCL
{ S7_Optimized_Access := 'TRUE' }
AUTHOR : Sachs
FAMILY : General
VERSION : 1.0
// stored: MemoryReserve 100, SetENOAutomatically false
   VAR_INPUT
      I_bEnable : Bool;
      I_bSeqMode : Bool;
      I_tTimeValue : Time;
   END_VAR
   VAR_OUTPUT
      O_bStart : Bool;
   END_VAR
   VAR
      ton_Delay { S7_SetPoint := 'True'} : TON_TIME;
      bStartdelay : Bool;
   END_VAR
BEGIN


   //***********************************************************************************************
   //下一步跳转模块/next step
   //***********************************************************************************************
   //延时条件
   IF #I_bEnable AND #I_bSeqMode AND (#ton_Delay.Q = FALSE OR #I_tTimeValue = t#0s) THEN
       #bStartdelay := TRUE;    
   END_IF;

   #ton_Delay(IN := #bStartdelay,
              PT := #I_tTimeValue);

   #O_bStart := #ton_Delay.Q;

   IF #ton_Delay.Q OR NOT #I_bEnable THEN
       #bStartdelay := FALSE; 
   END_IF;
END_FUNCTION_BLOCK

FUNCTION_BLOCK "CheckPositioningOrder"   // FB1, LAD
{ S7_Optimized_Access := 'TRUE' }
// stored: MemoryReserve 100, SetENOAutomatically false
   VAR_INPUT
      "V90Servo[3]" : Struct
         i : Int;
         nError : Int;
         nWarning : Int;
         nPositionListNo : Int := 1;
         Pos : "PosList";
         Point : Array[0..39] of Struct
            Start : Bool;
            Achieve : Bool;
         END_STRUCT;
      END_STRUCT;
   END_VAR
   VAR_OUTPUT
      HaveAxisStart : Bool;
      AxisStartNumber : Int;
   END_VAR
   VAR
      Index : Int;
   END_VAR
BEGIN

REGION Network 2 (SCL)
   FOR #Index := 0 TO 39 DO
       IF #"V90Servo[3]".Point[#Index].Start THEN
           #HaveAxisStart := true;
           #AxisStartNumber := #Index;
           EXIT;
       ELSE
           #HaveAxisStart := FALSE;
           #AxisStartNumber := 32767;
       END_IF;
   END_FOR;
END_REGION
END_FUNCTION_BLOCK

FUNCTION "块_1" : Void   // FC1, LAD
{ S7_Optimized_Access := 'TRUE' }
// stored: SetENOAutomatically false
BEGIN

REGION Network 2 (SCL)
   "CheckPositioningOrder_IDB"("V90Servo[3]":="ServoV90_DeviceCtl".V90Servo[3],
                               HaveAxisStart=>"DATA".HaveAxisStart,
                               AxisStartNumber=>"DATA".AxisStartNumber);

   //When the 382A1 card is stuck at step 130, change the process step to 100 and locate it again.
   //当382A1卡在 130步时,修改流程步去100再次定位
   IF    "DATA"."Forced modification"    AND
       "DATA".HaveAxisStart AND "DATA".AxisStartNumber <> 32767 AND
       "V90Servo_DB".Servo_382A1.sStep[1] = 130AND
       "V90Servo_DB".Servo_382A1.sErrorCode=0  AND
      // "ServoV90_A3".Auto.Pos["ServoV90_A3".Auto.Index].Pos<> "ServoV90_A3".Out.oActPosition
       "ServoV90_A3".Auto.Pos[6].Pos<> "ServoV90_A3".Out.oActPosition
   THEN
       "V90Servo_DB".Servo_382A1.sStep[1] := 100
       ;
   END_IF;
END_REGION
END_FUNCTION

FUNCTION_BLOCK "SINA_PARA_S"   // FB1821, SCL
{ S7_Optimized_Access := 'TRUE' }
AUTHOR : DRVDPS7
FAMILY : DRIVES
NAME : SINA_PAS
VERSION : 5.0
// stored: AutoNumber false, MemoryReserve 100, SetENOAutomatically false
   VAR_INPUT
      Start : Bool := 0;
      ReadWrite : Bool := 0;
      Parameter : Int := 1;
      Index : Int := 0;
      ValueWrite1 : Real := 0.0;
      ValueWrite2 : DInt := 0;
      AxisNo : Byte := 16#01;
      hardwareId : HW_IO := 0;
   END_VAR
   VAR_OUTPUT
      Ready : Bool := 0;
      Busy : Bool := 0;
      Done : Bool := 1;
      ValueRead1 : Real := 0.0;
      ValueRead2 : DInt := 0;
      Format : Byte := 16#00;
      ErrorNo : Word := 16#0000;
      Error : Bool := 0;
      ErrorId : DWord := 0;
      DiagId : Word := 16#0000;
   END_VAR
   VAR
      sbWrError : Bool := 0;
      sbWrDone : Bool := 0;
      sbRdError : Bool := 0;
      sbWrBusy : Bool := 0;
      sbRdBusy : Bool := 0;
      sbWrStart : Bool := 0;
      sbRdStart : Bool := 0;
      sbWrStart1 : Bool := 0;
      sbRdStart1 : Bool := 0;
      sbWrStart2 : Bool := 0;
      sbRdStart2 : Bool := 0;
      sbStart : Bool := 0;
      sbReady : Bool := 0;
      sbRead : Bool := 0;
      sbWrite : Bool := 0;
      sbParaNo : Bool := 0;
      sbBusy : Bool := 0;
      sbError : Bool := 0;
      sbDone : Bool := 0;
      syFormat : Byte := 16#00;
      syAxisNo : Byte := 0;
      siReqRef : Int := 0;
      siErrorId : Int := 0;
      siErrorCount : Int := 0;
      siMaxErrCount : Int := 12500;
      swParaError : Word := WORD#16#0000;
      sxReqParaMulti : Struct
         sxHeader : Struct
            syReqRef : Byte := 16#00;
            syReqId : Byte := 16#01;
            syAxisNo : Byte := 16#00;
            syParaNo : Byte := 16#00;
         END_STRUCT;
         sxParaAdress : Struct
            syAttr : Byte := 16#10;
            syElemNo : Byte := 16#01;
            siParaNo : Int := 0;
            siIndex : Int := 0;
         END_STRUCT;
      END_STRUCT;
      sxChaParaMulti : Struct
         sxHeader : Struct
            syReqRef : Byte := 16#00;
            syReqId : Byte := 16#02;
            syAxisNo : Byte := 16#00;
            syParaNo : Byte := 16#00;
         END_STRUCT;
         sxData : Array[1..12] of Byte;
      END_STRUCT;
      sxRespParaMulti : Struct
         sxHeader : Struct
            syReqRef : Byte := 16#00;
            syReqId : Byte := 16#00;
            syAxisNo : Byte := 16#00;
            syParaNo : Byte := 16#00;
         END_STRUCT;
         sxData : Array[1..6] of Byte;
      END_STRUCT;
      RDREC_1 { S7_SetPoint := 'True'} : RDREC;
      WRREC_1 { S7_SetPoint := 'True'} : WRREC;
      siLenHeader : Int := 4;
      siLenParaMulti : Int := 6;
      siLenChaPara : Int := 12;
   END_VAR
   VAR_TEMP
      piCount : Int;
      piPointer : Int;
      piLenTele : Int;
      piRetSFC : Int;
      pwWordHigh : Word;
      pwWordLow : Word;
      pwWord1 : Word;
      pwWord2 : Word;
      pdDWordHigh : DWord;
      pdDWordLow : DWord;
      pdStatus : DWord;
      pbValidSFB : Bool;
      piLenSFB : UInt;
      pwErrorNo : Word;
   END_VAR
BEGIN

   //=============================================================================
   //SIEMENS AG
   //(c)Copyright 2017 All Rights Reserved
   //-----------------------------------------------------------------------------
   // Library: DriveLib
   // Tested with: S7-1516-3 PN/DP V1.8
   // Engineering: TIA Portal V14
   // Restrictions: -
   // Requirements: S7-1200 / S7-1500
   // Functionality: read and write one parameter from/to a Sinamics
   //
   //=============================================================================

   // Auftrag "Parameter lesen" bzw. Auftrag "Parameter schreiben" wird nicht mehr ausgeführt
   IF NOT #sbBusy THEN
     #sbParaNo := TRUE;
     #syAxisNo := #AxisNo;
   END_IF;

   // Starten 
   IF #Start AND NOT #sbStart AND NOT #sbBusy THEN

     #sbReady := False;
     #sbError := False;
     #sbBusy := False;

     // Auftrag "Parameter lesen" erkennen
     IF NOT #ReadWrite THEN
       #sbRead := True;
       #sbWrStart := True;
       #sbRdStart := False;

       #sbWrite := False;
       #sbWrStart1 := False;
       #sbRdStart1 := False;
       #sbWrStart2 := False;
       #sbRdStart2 := False;

       // Referenzauftragsnummer erzeugen
       #siReqRef := #siReqRef + 1;

       // bei Überschreitung wieder zurücksetzen und von vorne (Wertebereich von 0-255)
       IF #siReqRef > 255 THEN
         #siReqRef := 0;
       END_IF;

       // Auftrag "Parameter schreiben" erkennen
     ELSE
       #sbWrite := True;
       #sbWrStart1 := True;
       #sbRdStart1 := False;
       #sbWrStart2 := False;
       #sbRdStart2 := False;

       #sbRead := False;
       #sbWrStart := False;
       #sbRdStart := False;

       // Referenzauftragsnummer erzeugen
       #siReqRef := #siReqRef + 1;

       // bei Überschreitung wieder zurücksetzen und von vorne (Wertebereich von 0-255)
       IF #siReqRef > 255 THEN
         #siReqRef := 0;
       END_IF;
     END_IF;

     // Fehler 4 und 5 wieder zurücknehmen
     IF (#siErrorId = 4) OR (#siErrorId = 5) THEN
       #sbError := False;
       #siErrorId := 0;
     END_IF;
   END_IF;

   // "Start commando" Flanke merken
   #sbStart := #Start;

   // Abbrechen
   IF NOT #Start THEN

     #siErrorCount := 0;
     // Schreib - oder Lesevorgang abbrechen
     #sbRead := False;
     #sbWrStart := False;
     #sbRdStart := False;

     #sbWrite := False;
     #sbWrStart1 := False;
     #sbRdStart1 := False;
     #sbWrStart2 := False;
     #sbRdStart2 := False;

     // Auftag ist noch beschäftigt => Fehler ausgeben
     IF #sbBusy THEN
       #sbError := True;
       #siErrorId := 4;
       #sbBusy := False;
     END_IF;
   END_IF;


   // Auftrag "Parameter lesen" wurde ausgelöst
   IF #sbParaNo AND #sbRead AND NOT #sbWrite THEN

     // Auftrag "Parameter lesen" vorbereiten und abschicken
     IF #sbWrStart THEN

       // Ablöschen des Sendepuffers
       // Parameternummer des Parameters 
       #sxReqParaMulti.sxParaAdress.siParaNo := 0;

       // Subindex des Parameters
       #sxReqParaMulti.sxParaAdress.siIndex := 0;

       // Auftrags-HEADER erstellen
       // Auftragsreferenz
       #sxReqParaMulti.sxHeader.syReqRef := INT_TO_BYTE(#siReqRef);

       // Auftragskennung 0x01=Request Parameters
       #sxReqParaMulti.sxHeader.syReqId := B#16#01;

       // Achse
       #sxReqParaMulti.sxHeader.syAxisNo := #syAxisNo;

       // Anzahl Parameter        
       #sxReqParaMulti.sxHeader.syParaNo := B#16#01;

       // Auftrags-PARAMETERADRESSE erstellen
       // Parameternummer des Parameters                                
       #sxReqParaMulti.sxParaAdress.siParaNo := #Parameter;

       // Subindex des Parameters
       #sxReqParaMulti.sxParaAdress.siIndex := #Index;

       // SCHREIBEN AZYKLISCH
       #piLenTele := #siLenHeader + #siLenParaMulti;
       #WRREC_1(REQ := True,                                // Startimpuls
                ID := #hardwareId,                         // Diagnoseadresse
                INDEX := 47,                                  // Rahmentyp
                LEN := INT_TO_UINT(#piLenTele),             // maximale Länge
                DONE => #sbWrDone,                           // Schreibauftrag beendet
                BUSY => #sbWrBusy,                           // Slave beschäftigt
                ERROR => #sbWrError,                          // Fehler beim Schreiben
                STATUS => #pdStatus,                           // Status[1] = Error => Status[2] Error Decode + Status[3] Error Code
                RECORD := #sxReqParaMulti);                    // Zeiger auf zu schreibenen Datensatzes

       // Ausgänge setzen
       #sbBusy := #sbWrBusy;
       #sbDone := #sbWrDone;

       // Fehler auswerten
       IF #sbWrError THEN

         // Fehlerstatus aus dem Doppelwort filtern und weitergeben                
         #pwWord1 := DWORD_TO_WORD(SHR(IN := (#pdStatus AND DW#16#FFFF00), N := 8));

         // Fehlerstatus setzen
         #siErrorId := 3;
         #DiagId := #pwWord1;

         //Temporärer Fehler: #pdStatus = 80A7, 80B5, 80C0, 80C1, 80C2, 80C3 oder 80C4 zulassen und nocheinmal versuchen
         IF NOT (#pwWord1 = DW#16#80A7) AND NOT (#pwWord1 = DW#16#80B5) AND NOT (#pwWord1 = DW#16#80C0) AND
           NOT (#pwWord1 = DW#16#80C1) AND NOT (#pwWord1 = DW#16#80C2) AND NOT (#pwWord1 = DW#16#80C3) AND
           NOT (#pwWord1 = DW#16#80C4) THEN

           // Wiederholungsauftrag wieder zurücknehmen 
           #sbWrStart := False;
           #sbRdStart := False;
           #sbRead := False;

           // Fehler ausgeben 
           #sbError := #sbWrError;

         ELSE
           // Fehlerwiederholauftrag ??                   
           IF #siErrorCount = #siMaxErrCount THEN

             // Wiederholungsauftrag wieder zurücknehmen
             #sbWrStart := False;
             #sbRdStart := False;
             #sbRead := False;

             //Fehlerzähler zurücksetzen
             #siErrorCount := 0;


             // Fehler ausgeben 
             #sbError := #sbWrError;

             // nix tun bis Zähler überläuft
           ELSE
             #siErrorCount := #siErrorCount + 1;
           END_IF;
         END_IF;

         // kein Fehler beim SCHEIBEN AZYKLISCH und Auftrag fertig 
       ELSIF NOT #sbWrBusy AND #sbWrDone THEN

         // Fehlerkennung zurücknehmen
         IF #siErrorId = 3 THEN
           #siErrorId := 0;
           #sbError := False;
         END_IF;

         #DiagId := W#16#00;

         // Schreibauftrag fertig melden und Leseantrag anstossen
         #sbWrStart := False;
         #sbRdStart := True;
       END_IF;
     END_IF; // Auftrag "Parameter lesen" vorbereiten und abschicken

     // vom Auftrag "Parameter lesen" die Antwort abwarten und dann auswerten
     IF #sbRdStart THEN

       // Ablöschen des Empfangspuffers
       #sxRespParaMulti.sxHeader.syReqRef := B#16#00;
       #sxRespParaMulti.sxHeader.syReqId := B#16#00;
       #sxRespParaMulti.sxHeader.syAxisNo := B#16#00;
       #sxRespParaMulti.sxHeader.syParaNo := B#16#00;

       FOR #piCount := 1 TO #siLenParaMulti DO
         #sxRespParaMulti.sxData[#piCount] := B#16#00;
       END_FOR;

       // LESEN AZYKLISCH
       #piLenTele := #siLenHeader + #siLenParaMulti;
       #RDREC_1(REQ := True,                                // Startimpuls
                ID := #hardwareId,                         // Diagnoseadresse        
                INDEX := 47,                                  // Rahmentyp           
                MLEN := INT_TO_UINT(#piLenTele),             // maximale Länge
                VALID => #pbValidSFB,                         // neuer Datensatz empfangen und gültig   
                BUSY => #sbRdBusy,                           // Slave beschäftigt
                ERROR => #sbRdError,                          // Fehler beim Schreiben
                STATUS => #pdStatus,                           // Status[1] = Error => Status[2] Error Decode + Status[3] Error Code 
                LEN => #piLenSFB,                           // Länge des gelesenen Datensatzes
                RECORD := #sxRespParaMulti);                   // Zeiger auf gelesenen Datensatz

       // Ausgänge setzen
       #sbBusy := #sbRdBusy;
       #sbDone := #pbValidSFB;

       // Fehler auswerten
       IF #sbRdError THEN
         // Fehlerstatus aus dem Doppelwort filtern und weitergeben                
         #pwWord1 := DWORD_TO_WORD(SHR(IN := (#pdStatus AND DW#16#FFFF00), N := 8));

         // Fehlerstatus setzen
         #siErrorId := 3;
         #DiagId := #pwWord1;

         //Temporärer Fehler: #pdStatus = 80A7, 80B5, 80C0, 80C1, 80C2, 80C3 oder 80C4 zulassen und nocheinmal versuchen
         IF NOT (#pwWord1 = DW#16#80A7) AND NOT (#pwWord1 = DW#16#80B5) AND NOT (#pwWord1 = DW#16#80C0) AND
           NOT (#pwWord1 = DW#16#80C1) AND NOT (#pwWord1 = DW#16#80C2) AND NOT (#pwWord1 = DW#16#80C3) AND
           NOT (#pwWord1 = DW#16#80C4) THEN

           // Wiederholungsauftrag wieder zurücknehmen  
           #sbWrStart := False;
           #sbRdStart := False;
           #sbRead := False;

           // Fehler ausgeben 
           #sbError := #sbRdError;

         ELSE
           // Fehlerwiederholauftrag ??                   
           IF #siErrorCount = #siMaxErrCount THEN

             // Wiederholungsauftrag wieder zurücknehmen
             #sbWrStart := False;
             #sbRdStart := False;
             #sbRead := False;

             //Fehlerzähler zurücksetzen
             #siErrorCount := 0;


             // Fehler ausgeben 
             #sbError := #sbRdError;

             // nix tun bis Zähler überläuft
           ELSE
             #siErrorCount := #siErrorCount + 1;
           END_IF;
         END_IF;

         // Fehler : die Auftragsreferenz der Antwort übertimmt nicht mit der Auftragsreferenz der Anfrage überein
       ELSIF NOT (#siReqRef = BYTE_TO_INT(#sxRespParaMulti.sxHeader.syReqRef)) AND NOT #sbRdBusy AND #pbValidSFB THEN
         #siErrorId := 1;
         #sbError := True;
         #sbDone := False;

         // Wiederholungsauftrag wieder zurücknehmen  
         #sbWrStart := False;
         #sbRdStart := False;
         #sbRead := False;

         // Fehler : falsche Auftragskennung zurück erhalten    
       ELSIF NOT (#sxRespParaMulti.sxHeader.syReqId = B#16#81 OR #sxRespParaMulti.sxHeader.syReqId = B#16#01) AND
         NOT #sbRdBusy AND #pbValidSFB THEN
         #siErrorId := 1;
         #sbError := True;
         #sbDone := False;

         // Wiederholungsauftrag wieder zurücknehmen  
         #sbWrStart := False;
         #sbRdStart := False;
         #sbRead := False;

         // Fehler : die angeforderte Anzahl Parameter entspricht nicht der übermittelten Anzahl Parameter überein
       ELSIF NOT (#sxRespParaMulti.sxHeader.syParaNo = B#16#01) AND NOT #sbRdBusy AND #pbValidSFB THEN
         #siErrorId := 1;
         #sbError := True;
         #sbDone := False;

         // Wiederholungsauftrag wieder zurücknehmen  
         #sbWrStart := False;
         #sbRdStart := False;
         #sbRead := False;

         // Fehler : die Achse entspricht nicht der übergebenen Achse
       ELSIF NOT (#syAxisNo = #sxRespParaMulti.sxHeader.syAxisNo) AND NOT #sbRdBusy AND #pbValidSFB THEN
         #siErrorId := 1;
         #sbError := True;
         #sbDone := False;

         // Wiederholungsauftrag wieder zurücknehmen  
         #sbWrStart := False;
         #sbRdStart := False;
         #sbRead := False;

         // kein Fehler beim LESEN AZYKLISCH und Auftrag fertig 
       ELSIF NOT #sbRdBusy AND #pbValidSFB THEN

         // die angefragten Parameter auswerten und im Puffer abspeichern

         // ermitteltes Format des Parameters abspeichern
         #syFormat := #sxRespParaMulti.sxData[1];

         // Format = Error ? = > gesendeter Parameter fehlerhaft
         IF (BYTE_TO_INT(#sxRespParaMulti.sxData[1]) = 68) THEN

           // Format = Error, zwei Bytes zu übermittelten Fehlernummer zusammenfassen
           #pwWordHigh := SHL(IN := BYTE_TO_WORD(#sxRespParaMulti.sxData[3]), N := 8);
           #pwWordLow := BYTE_TO_WORD(#sxRespParaMulti.sxData[4]);

           #sbError := True;

           // ermittelte Fehlernummer im Puffer abspeichern
           #ErrorNo := #pwWordHigh XOR #pwWordLow;

           // Die Fehlerhaftigkeit des erkannten Parameter in der Fehlernummer eintragen   
           #swParaError := #swParaError OR W#16#01;

           // Format = Byte ? = > gesendeter Parameter ein Byte lang ohne Vorzeichen
         ELSIF (#sxRespParaMulti.sxData[1] = B#16#41) OR (#sxRespParaMulti.sxData[1] = B#16#05) THEN

           // ermittelter Parameterwert eintragen (Byte) 
           #ValueRead1 := USINT_TO_REAL(BYTE_TO_USINT(#sxRespParaMulti.sxData[3]));
           #ValueRead2 := 0;

           // ermittelte Fehlernummer im Puffer zurücksetzen
           #ErrorNo := W#16#00;

           // Die Fehlerhaftigkeit des erkannten Parameter in der Fehlernummer löschen   
           #swParaError := #swParaError AND W#16#FFFE;

           // Format = Byte ? = > gesendeter Parameter ein Byte lang mit Vorzeichen
         ELSIF (#sxRespParaMulti.sxData[1] = B#16#02) THEN

           // ermittelter Parameterwert eintragen (Byte) 
           #ValueRead1 := SINT_TO_REAL(BYTE_TO_SINT(#sxRespParaMulti.sxData[3]));
           #ValueRead2 := 0;

           // ermittelte Fehlernummer im Puffer zurücksetzen
           #ErrorNo := W#16#00;

           // Die Fehlerhaftigkeit des erkannten Parameter in der Fehlernummer löschen   
           #swParaError := #swParaError AND W#16#FFFE;

           // Format = Word ? = > gesendeter Parameter zwei Bytes lang ohne Vorzeichen
         ELSIF (#sxRespParaMulti.sxData[1] = B#16#42) OR (#sxRespParaMulti.sxData[1] = B#16#06)
           OR (#sxRespParaMulti.sxData[1] = B#16#0A) THEN

           // Format = Word, zwei Bytes zu übermitteltem Parameterwert zusammenfassen
           #pwWordHigh := SHL(IN := BYTE_TO_WORD(#sxRespParaMulti.sxData[3]), N := 8);
           #pwWordLow := BYTE_TO_WORD(#sxRespParaMulti.sxData[4]);
           #pwWord1 := #pwWordHigh XOR #pwWordLow;

           // ermittelter Parameterwert eintragen (Word)
           #ValueRead1 := UINT_TO_REAL(WORD_TO_UINT(#pwWord1));
           #ValueRead2 := 0;

           // ermittelte Fehlernummer im Puffer zurücksetzen
           #ErrorNo := W#16#00;

           // Die Fehlerhaftigkeit des erkannten Parameter in der Fehlernummer löschen   
           #swParaError := #swParaError AND W#16#FFFE;

           // Format = Word ? = > gesendeter Parameter zwei Bytes lang mit Vorzeichen
         ELSIF (#sxRespParaMulti.sxData[1] = B#16#03) THEN

           // Format = Word, zwei Bytes zu übermitteltem Parameterwert zusammenfassen
           #pwWordHigh := SHL(IN := BYTE_TO_WORD(#sxRespParaMulti.sxData[3]), N := 8);
           #pwWordLow := BYTE_TO_WORD(#sxRespParaMulti.sxData[4]);
           #pwWord1 := #pwWordHigh XOR #pwWordLow;

           // ermittelter Parameterwert eintragen (Word)
           #ValueRead1 := INT_TO_REAL(WORD_TO_INT(#pwWord1));
           #ValueRead2 := 0;

           // ermittelte Fehlernummer im Puffer zurücksetzen
           #ErrorNo := W#16#00;

           // Die Fehlerhaftigkeit des erkannten Parameter in der Fehlernummer löschen   
           #swParaError := #swParaError AND W#16#FFFE;

           // Format = Double Word ? = > gesendeter Parameter vier Bytes lang ohne Vorzeichen
         ELSIF (#sxRespParaMulti.sxData[1] = B#16#43) OR (#sxRespParaMulti.sxData[1] = B#16#07) OR
           (#sxRespParaMulti.sxData[1] = B#16#0D) THEN

           // Format = Double Word, vier Bytes zu übermitteltem Parameterwert zusammenfassen
           #pwWordHigh := SHL(IN := BYTE_TO_WORD(#sxRespParaMulti.sxData[3]), N := 8);
           #pwWordLow := BYTE_TO_WORD(#sxRespParaMulti.sxData[4]);
           #pwWord1 := #pwWordHigh XOR #pwWordLow;

           #pwWordHigh := SHL(IN := BYTE_TO_WORD(#sxRespParaMulti.sxData[5]), N := 8);
           #pwWordLow := BYTE_TO_WORD(#sxRespParaMulti.sxData[6]);
           #pwWord2 := #pwWordHigh XOR #pwWordLow;

           #pdDWordHigh := SHL(IN := WORD_TO_DWORD(#pwWord1), N := 16);
           #pdDWordLow := WORD_TO_DWORD(#pwWord2);

           // ermittelter Parameterwert eintragen (Word)
           #ValueRead1 := 0.0;
           #ValueRead2 := DWORD_TO_DINT(#pdDWordHigh XOR #pdDWordLow);

           // ermittelte Fehlernummer im Puffer zurücksetzen
           #ErrorNo := W#16#00;

           // Die Fehlerhaftigkeit des erkannten Parameter in der Fehlernummer löschen   
           #swParaError := #swParaError AND W#16#FFFE;

           // Format = Double Word ? = > gesendeter Parameter vier Bytes lang mit Vorzeichen
         ELSIF (#sxRespParaMulti.sxData[1] = B#16#04) THEN

           // Format = Double Word, vier Bytes zu übermitteltem Parameterwert zusammenfassen
           #pwWordHigh := SHL(IN := BYTE_TO_WORD(#sxRespParaMulti.sxData[3]), N := 8);
           #pwWordLow := BYTE_TO_WORD(#sxRespParaMulti.sxData[4]);
           #pwWord1 := #pwWordHigh XOR #pwWordLow;

           #pwWordHigh := SHL(IN := BYTE_TO_WORD(#sxRespParaMulti.sxData[5]), N := 8);
           #pwWordLow := BYTE_TO_WORD(#sxRespParaMulti.sxData[6]);
           #pwWord2 := #pwWordHigh XOR #pwWordLow;

           #pdDWordHigh := SHL(IN := WORD_TO_DWORD(#pwWord1), N := 16);
           #pdDWordLow := WORD_TO_DWORD(#pwWord2);

           // ermittelter Parameterwert eintragen (Word)
           #ValueRead1 := 0.0;
           #ValueRead2 := DWORD_TO_DINT(#pdDWordHigh XOR #pdDWordLow);

           // ermittelte Fehlernummer im Puffer zurücksetzen
           #ErrorNo := W#16#00;

           // Die Fehlerhaftigkeit des erkannten Parameter in der Fehlernummer löschen   
           #swParaError := #swParaError AND W#16#FFFE;

           // Format = Double Word ? = > gesendeter Parameter vier Bytes lang (FloatingPoint)
         ELSIF (#sxRespParaMulti.sxData[1] = B#16#08) THEN

           // Format = Double Word, vier Bytes zu übermitteltem Parameterwert zusammenfassen
           #pwWordHigh := SHL(IN := BYTE_TO_WORD(#sxRespParaMulti.sxData[3]), N := 8);
           #pwWordLow := BYTE_TO_WORD(#sxRespParaMulti.sxData[4]);
           #pwWord1 := #pwWordHigh XOR #pwWordLow;

           #pwWordHigh := SHL(IN := BYTE_TO_WORD(#sxRespParaMulti.sxData[5]), N := 8);
           #pwWordLow := BYTE_TO_WORD(#sxRespParaMulti.sxData[6]);
           #pwWord2 := #pwWordHigh XOR #pwWordLow;

           #pdDWordHigh := SHL(IN := WORD_TO_DWORD(#pwWord1), N := 16);
           #pdDWordLow := WORD_TO_DWORD(#pwWord2);

           // ermittelter Parameterwert eintragen (Word)
           #ValueRead1 := DWORD_TO_REAL(#pdDWordHigh XOR #pdDWordLow);
           #ValueRead2 := 0;

           // ermittelte Fehlernummer im Puffer zurücksetzen
           #ErrorNo := W#16#00;

           // Die Fehlerhaftigkeit des erkannten Parameter in der Fehlernummer löschen   
           #swParaError := #swParaError AND W#16#FFFE;

           // Unbekanter Datentyp
         ELSE

           #siErrorId := 5;
           #sbError := True;
           #sbDone := False;
           // Die Fehlerhaftigkeit des erkannten Parameter in der Fehlernummer eintragen   
           #swParaError := #swParaError OR W#16#01;

         END_IF;

         // Fehlerkennung zurücknehmen
         IF (#siErrorId = 3) OR (#siErrorId = 1) THEN
           #siErrorId := 0;
           #sbError := False;
         END_IF;

         #DiagId := W#16#00;

         // Auftrag : Parameter lesen ist abgeschlossen
         #sbRdStart := False;
         #sbRead := False;
       END_IF; // kein Fehler beim LESEN AZYKLISCH und Auftrag fertig 
     END_IF; // vom Auftrag "Parameter lesen" die Antwort abwarten und dann auswerten 
   END_IF; // Auftrag "Parameter lesen" wurde ausgelöst

   // Auftrag "Parameter schreiben" wurde ausgelöst
   IF #sbParaNo AND NOT #sbRead AND #sbWrite THEN

     // Auftrag "Parameter schreiben" bzw. "ändern" besteht aus zwei Aufträgen
     // 1. Teilauftrag "Parameter lesen"
     // 2. Teilauftrag "Parameter schreiben bzw. ändern"

     // 1. Teilauftrag "Parameter lesen" vorbereiten und abschicken
     IF #sbWrStart1 THEN

       // Ablöschen des Sendepuffers
       // Parameternummer des Parameters 
       #sxReqParaMulti.sxParaAdress.siParaNo := 0;

       // Subindex des Parameters
       #sxReqParaMulti.sxParaAdress.siIndex := 0;

       // Auftrags-HEADER erstellen
       // Auftragsreferenz
       #sxReqParaMulti.sxHeader.syReqRef := INT_TO_BYTE(#siReqRef);

       // Auftragskennung 0x01=Request Parameters
       #sxReqParaMulti.sxHeader.syReqId := B#16#01;

       // Achse
       #sxReqParaMulti.sxHeader.syAxisNo := #syAxisNo;

       // Anzahl Parameter        
       #sxReqParaMulti.sxHeader.syParaNo := B#16#01;

       // Auftrags-PARAMETERADRESSE erstellen
       // Parameternummer des Parameters                                
       #sxReqParaMulti.sxParaAdress.siParaNo := #Parameter;

       // Subindex des Parameters
       #sxReqParaMulti.sxParaAdress.siIndex := #Index;

       // SCHREIBEN AZYKLISCH
       #piLenTele := #siLenHeader + #siLenParaMulti;
       #WRREC_1(REQ := True,                                // Startimpuls
                ID := #hardwareId,                         // Diagnoseadresse
                INDEX := 47,                                  // Rahmentyp
                LEN := INT_TO_UINT(#piLenTele),             // maximale Länge
                DONE => #sbWrDone,                           // Schreibauftrag beendet
                BUSY => #sbWrBusy,                           // Slave beschäftigt
                ERROR => #sbWrError,                          // Fehler beim Schreiben
                STATUS => #pdStatus,                           // Status[1] = Error => Status[2] Error Decode + Status[3] Error Code
                RECORD := #sxReqParaMulti);                    // Zeiger auf zu schreibenen Datensatz

       // Ausgänge setzen
       #sbBusy := #sbWrBusy;
       #sbDone := #sbWrDone;

       // Fehler auswerten
       IF #sbWrError THEN

         // Fehlerstatus aus dem Doppelwort filtern und weitergeben                
         #pwWord1 := DWORD_TO_WORD(SHR(IN := (#pdStatus AND DW#16#FFFF00), N := 8));

         // Fehlerstatus setzen
         #siErrorId := 3;
         #DiagId := #pwWord1;

         //Temporärer Fehler: #pdStatus = 80A7, 80B5, 80C0, 80C1, 80C2, 80C3 oder 80C4 zulassen und nocheinmal versuchen
         IF NOT (#pwWord1 = DW#16#80A7) AND NOT (#pwWord1 = DW#16#80B5) AND NOT (#pwWord1 = DW#16#80C0) AND
           NOT (#pwWord1 = DW#16#80C1) AND NOT (#pwWord1 = DW#16#80C2) AND NOT (#pwWord1 = DW#16#80C3) AND
           NOT (#pwWord1 = DW#16#80C4) THEN

           // Wiederholungsauftrag wieder zurücknehmen
           #sbWrStart1 := False;
           #sbRdStart1 := False;
           #sbWrite := False;

           // Fehler ausgeben 
           #sbError := #sbWrError;

         ELSE
           // Fehlerwiederholauftrag ??                   
           IF #siErrorCount = #siMaxErrCount THEN

             // Wiederholungsauftrag wieder zurücknehmen
             #sbWrStart1 := False;
             #sbRdStart1 := False;
             #sbWrite := False;

             //Fehlerzähler zurücksetzen
             #siErrorCount := 0;


             // Fehler ausgeben 
             #sbError := #sbWrError;
             // nix tun bis Zähler überläuft
           ELSE
             #siErrorCount := #siErrorCount + 1;
           END_IF;
         END_IF;

         // kein Fehler beim SCHEIBEN AZYKLISCH und Auftrag fertig 
       ELSIF NOT #sbWrBusy AND #sbWrDone THEN

         // Fehlerkennung zurücknehmen
         IF (#siErrorId = 3) THEN
           #siErrorId := 0;
           #sbError := False;
         END_IF;

         #DiagId := W#16#00;

         // Schreibauftrag fertig melden und Leseantrag anstossen
         #sbWrStart1 := False;
         #sbRdStart1 := True;
       END_IF;
     END_IF; // 1. Teilauftrag "Parameter lesen" vorbereiten und abschicken

     // vom 1. Teilauftrag "Parameter lesen" die Antwort abwarten und dann auswerten
     IF #sbRdStart1 THEN

       // Ablöschen des Empfangspuffers
       #sxRespParaMulti.sxHeader.syReqRef := B#16#00;
       #sxRespParaMulti.sxHeader.syReqId := B#16#00;
       #sxRespParaMulti.sxHeader.syAxisNo := B#16#00;
       #sxRespParaMulti.sxHeader.syParaNo := B#16#00;

       FOR #piCount := 1 TO #siLenParaMulti DO
         #sxRespParaMulti.sxData[#piCount] := B#16#00;
       END_FOR;

       // LESEN AZYKLISCH
       #piLenTele := #siLenHeader + #siLenParaMulti;
       #RDREC_1(REQ := True,                                // Startimpuls
                ID := #hardwareId,                         // Diagnoseadresse        
                INDEX := 47,                                  // Rahmentyp           
                MLEN := INT_TO_UINT(#piLenTele),             // maximale Länge
                VALID => #pbValidSFB,                         // neuer Datensatz empfangen und gültig      
                BUSY => #sbRdBusy,                           // Slave beschäftigt
                ERROR => #sbRdError,                          // Fehler beim Schreiben
                STATUS => #pdStatus,                           // Status[1] = Error => Status[2] Error Decode + Status[3] Error Code 
                LEN => #piLenSFB,                           // Länge des gelesenen Datensatzes
                RECORD := #sxRespParaMulti);                   // Zeiger auf gelesenen Datensatz

       // Ausgänge setzen
       #sbBusy := #sbRdBusy;
       #sbDone := #pbValidSFB;

       // Fehler auswerten
       IF #sbRdError THEN
         // Fehlerstatus aus dem Doppelwort filtern und weitergeben                
         #pwWord1 := DWORD_TO_WORD(SHR(IN := (#pdStatus AND DW#16#FFFF00), N := 8));

         // Fehlerstatus setzen
         #siErrorId := 3;
         #DiagId := #pwWord1;

         //Temporärer Fehler: #pdStatus = 80A7, 80B5, 80C0, 80C1, 80C2, 80C3 oder 80C4 zulassen und nocheinmal versuchen
         IF NOT (#pwWord1 = DW#16#80A7) AND NOT (#pwWord1 = DW#16#80B5) AND NOT (#pwWord1 = DW#16#80C0) AND
           NOT (#pwWord1 = DW#16#80C1) AND NOT (#pwWord1 = DW#16#80C2) AND NOT (#pwWord1 = DW#16#80C3) AND
           NOT (#pwWord1 = DW#16#80C4) THEN

           // Wiederholungsauftrag wieder zurücknehmen
           #sbWrStart1 := False;
           #sbRdStart1 := False;
           #sbWrite := False;

           // Fehler ausgeben 
           #sbError := #sbRdError;

         ELSE
           // Fehlerwiederholauftrag ??                   
           IF #siErrorCount = #siMaxErrCount THEN

             // Wiederholungsauftrag wieder zurücknehmen
             #sbWrStart1 := False;
             #sbRdStart1 := False;
             #sbWrite := False;

             //Fehlerzähler zurücksetzen
             #siErrorCount := 0;


             // Fehler ausgeben 
             #sbError := #sbRdError;

             // nix tun bis Zähler überläuft
           ELSE
             #siErrorCount := #siErrorCount + 1;
           END_IF;
         END_IF;

         // Fehler : die Auftragsreferenz der Antwort übertimmt nicht mit der Auftragsreferenz der Anfrage überein
       ELSIF NOT (#siReqRef = BYTE_TO_INT(#sxRespParaMulti.sxHeader.syReqRef)) AND NOT #sbRdBusy AND #pbValidSFB THEN
         #siErrorId := 1;
         #sbError := True;
         #sbDone := False;

         // Wiederholungsauftrag wieder zurücknehmen
         #sbWrStart1 := False;
         #sbRdStart1 := False;
         #sbWrite := False;

         // Fehler : falsche Auftragskennung zurück erhalten    
       ELSIF NOT (#sxRespParaMulti.sxHeader.syReqId = B#16#81 OR #sxRespParaMulti.sxHeader.syReqId = B#16#01) AND
         NOT #sbRdBusy AND #pbValidSFB THEN
         #siErrorId := 1;
         #sbError := True;
         #sbDone := False;

         // Wiederholungsauftrag wieder zurücknehmen
         #sbWrStart1 := False;
         #sbRdStart1 := False;
         #sbWrite := False;

         // Fehler : die angeforderte Anzahl Parameter entspricht nicht der übermittelten Anzahl Parameter überein
       ELSIF NOT (#sxRespParaMulti.sxHeader.syParaNo = B#16#01) AND NOT #sbRdBusy AND #pbValidSFB THEN
         #siErrorId := 1;
         #sbError := True;
         #sbDone := False;

         // Wiederholungsauftrag wieder zurücknehmen
         #sbWrStart1 := False;
         #sbRdStart1 := False;
         #sbWrite := False;

         // Fehler : die Achse entspricht nicht der übergebenen Achse
       ELSIF NOT (#syAxisNo = #sxRespParaMulti.sxHeader.syAxisNo) AND NOT #sbRdBusy AND #pbValidSFB THEN
         #siErrorId := 1;
         #sbError := True;
         #sbDone := False;

         // Wiederholungsauftrag wieder zurücknehmen
         #sbWrStart1 := False;
         #sbRdStart1 := False;
         #sbWrite := False;

         // kein Fehler beim LESEN AZYKLISCH und Auftrag fertig 
       ELSIF NOT #sbRdBusy AND #pbValidSFB THEN

         // die angefragten Parameter auswerten und im Puffer abspeichern
         // ermitteltes Format des Parameters abspeichern
         #syFormat := #sxRespParaMulti.sxData[1];

         // Format = Error ? = > gesendeter Parameter fehlerhaft
         IF (BYTE_TO_INT(#sxRespParaMulti.sxData[1]) = 68) THEN

           // Format = Error, zwei Bytes zu übermittelten Fehlernummer zusammenfassen
           #pwWordHigh := SHL(IN := BYTE_TO_WORD(#sxRespParaMulti.sxData[3]), N := 8);
           #pwWordLow := BYTE_TO_WORD(#sxRespParaMulti.sxData[4]);

           #sbError := True;

           // ermittelte Fehlernummer im Puffer abspeichern
           #ErrorNo := #pwWordHigh XOR #pwWordLow;

           // Die Fehlerhaftigkeit des erkannten Parameter in der Fehlernummer eintragen   
           #swParaError := #swParaError OR W#16#01;

           // Format = Byte ? = > gesendeter Parameter ein Byte lang
         ELSIF (#sxRespParaMulti.sxData[1] = B#16#41) OR
           (#sxRespParaMulti.sxData[1] = B#16#02) OR (#sxRespParaMulti.sxData[1] = B#16#05) THEN

           // ermittelte Fehlernummer im Puffer zurücksetzen
           #ErrorNo := W#16#00;

           // Die Fehlerhaftigkeit des erkannten Parameter in der Fehlernummer löschen   
           #swParaError := #swParaError AND W#16#FFFE;

           // Format = Word ? = > gesendeter Parameter zwei Bytes lang
         ELSIF (#sxRespParaMulti.sxData[1] = B#16#42) OR (#sxRespParaMulti.sxData[1] = B#16#03)
           OR (#sxRespParaMulti.sxData[1] = B#16#06) OR (#sxRespParaMulti.sxData[1] = B#16#0A) THEN

           // ermittelte Fehlernummer im Puffer zurücksetzen
           #ErrorNo := W#16#00;

           // Die Fehlerhaftigkeit des erkannten Parameter in der Fehlernummer löschen   
           #swParaError := #swParaError AND W#16#FFFE;


           // Format = Double Word ? = > gesendeter Parameter vier Bytes lang
         ELSIF (#sxRespParaMulti.sxData[1] = B#16#43) OR (#sxRespParaMulti.sxData[1] = B#16#04) OR
           (#sxRespParaMulti.sxData[1] = B#16#07) OR (#sxRespParaMulti.sxData[1] = B#16#08) OR
           (#sxRespParaMulti.sxData[1] = B#16#0D) THEN

           // ermittelte Fehlernummer im Puffer zurücksetzen
           #ErrorNo := W#16#00;

           // Die Fehlerhaftigkeit des erkannten Parameter in der Fehlernummer löschen   
           #swParaError := #swParaError AND W#16#FFFE;

           // Unbekanter Datentyp
         ELSE

           #siErrorId := 5;
           #sbError := True;
           #sbDone := False;
           // Die Fehlerhaftigkeit des erkannten Parameter in der Fehlernummer eintragen   
           #swParaError := #swParaError OR W#16#01;

         END_IF;

         // Fehlerkennung zurücknehmen
         IF (#siErrorId = 3) OR (#siErrorId = 1) THEN
           #siErrorId := 0;
           #sbError := False;
         END_IF;

         #DiagId := W#16#00;

         // 1. Teilauftrag "Parameter lesen" ist abgeschlossen
         #sbRdStart1 := False;

         // einer der gesendeten Parameter ist fehlerhaft => Abbruch, kein "Parameter schreiben" erforderlich
         IF (#swParaError = W#16#00) THEN
           #sbWrStart2 := True;
         ELSE
           #sbWrStart2 := False;
         END_IF;
       END_IF; // kein Fehler beim LESEN AZYKLISCH und Auftrag fertig 
     END_IF; // vom 1. Teilauftrag "Parameter lesen" die Antwort abwarten und dann auswerten 

     // 2. Teilauftrag "Parameter schreiben bzw. ändern" vorbereiten und abschicken
     IF #sbWrStart2 THEN

       // Ablöschen des Sendepuffers            
       FOR #piCount := 1 TO #siLenChaPara DO
         // Parameteradresse und Parameterwert des Parameters 
         #sxChaParaMulti.sxData[#piCount] := B#16#00;
       END_FOR;

       // Auftrags-HEADER erstellen
       // Auftragsreferenz
       #sxChaParaMulti.sxHeader.syReqRef := INT_TO_BYTE(#siReqRef);

       // Auftragskennung 0x01=Request Parameters | 0x02=Change Parameters
       #sxChaParaMulti.sxHeader.syReqId := B#16#02;

       // Achse
       #sxChaParaMulti.sxHeader.syAxisNo := #syAxisNo;

       // Anzahl Parameter        
       #sxChaParaMulti.sxHeader.syParaNo := B#16#01;

       // Auftrags-PARAMETERADRESSE erstellen                
       // Attribute of parameters (0x10=Value, 0x30=Text)
       #sxChaParaMulti.sxData[1] := B#16#10;

       // No. of elements (DEC: for single elements=1) 
       #sxChaParaMulti.sxData[2] := B#16#01;

       // Parameternummer des Parameters                                
       #sxChaParaMulti.sxData[4] := INT_TO_BYTE(#Parameter);
       #sxChaParaMulti.sxData[3] := WORD_TO_BYTE(SHR(IN := INT_TO_WORD(#Parameter), N := 8));

       // Subindex des Parameters
       #sxChaParaMulti.sxData[6] := INT_TO_BYTE(#Index);
       #sxChaParaMulti.sxData[5] := WORD_TO_BYTE(SHR(IN := INT_TO_WORD(#Index), N := 8));

       // Auftrags-PARAMETERVALUE erstellen    
       // Format (BYTE, WORD, DWORD des Parameterwert übergeben
       #sxChaParaMulti.sxData[7] := #syFormat;

       // Number of value
       #sxChaParaMulti.sxData[8] := B#16#01;

       // Value of parameter in Bytes
       IF (#syFormat = B#16#41) OR
         (#syFormat = B#16#02) OR (#syFormat = B#16#05) THEN

         #sxChaParaMulti.sxData[9] := WORD_TO_BYTE(DWORD_TO_WORD(DINT_TO_DWORD(REAL_TO_DINT(#ValueWrite1))));
         #sxChaParaMulti.sxData[10] := 16#00;  //WORD_TO_BYTE(DWORD_TO_WORD(SHR(IN := DINT_TO_DWORD(REAL_TO_DINT(#ValueWrite1)), N := 8)));

         // Value of parameter in Word
       ELSIF (#syFormat = B#16#42) OR (#syFormat = B#16#03) OR
         (#syFormat = B#16#06) OR (#syFormat = B#16#0A) THEN

         #sxChaParaMulti.sxData[10] := WORD_TO_BYTE(DWORD_TO_WORD(DINT_TO_DWORD(REAL_TO_DINT(#ValueWrite1))));
         #sxChaParaMulti.sxData[9] := WORD_TO_BYTE(DWORD_TO_WORD(SHR(IN := DINT_TO_DWORD(REAL_TO_DINT(#ValueWrite1)), N := 8)));

         // Value of parameter in DWord    
       ELSIF (#syFormat = B#16#43) OR (#syFormat = B#16#04) OR
         (#syFormat = B#16#07) OR (#syFormat = B#16#0D) THEN

         #sxChaParaMulti.sxData[12] := WORD_TO_BYTE(DWORD_TO_WORD(DINT_TO_DWORD(#ValueWrite2)));
         #sxChaParaMulti.sxData[11] := WORD_TO_BYTE(DWORD_TO_WORD(SHR(IN := DINT_TO_DWORD(#ValueWrite2), N := 8)));
         #sxChaParaMulti.sxData[10] := WORD_TO_BYTE(DWORD_TO_WORD(SHR(IN := DINT_TO_DWORD(#ValueWrite2), N := 16)));
         #sxChaParaMulti.sxData[9] := WORD_TO_BYTE(DWORD_TO_WORD(SHR(IN := DINT_TO_DWORD(#ValueWrite2), N := 24)));


         // Value of parameter in DWord (FloatingPoint)   
       ELSIF (#syFormat = B#16#08) THEN

         #sxChaParaMulti.sxData[12] := WORD_TO_BYTE(DWORD_TO_WORD(REAL_TO_DWORD(#ValueWrite1)));
         #sxChaParaMulti.sxData[11] := WORD_TO_BYTE(DWORD_TO_WORD(SHR(IN := REAL_TO_DWORD(#ValueWrite1), N := 8)));
         #sxChaParaMulti.sxData[10] := WORD_TO_BYTE(DWORD_TO_WORD(SHR(IN := REAL_TO_DWORD(#ValueWrite1), N := 16)));
         #sxChaParaMulti.sxData[9] := WORD_TO_BYTE(DWORD_TO_WORD(SHR(IN := REAL_TO_DWORD(#ValueWrite1), N := 24)));

       END_IF;

       // SCHREIBEN AZYKLISCH
       #piLenTele := #siLenHeader + #siLenChaPara;
       #WRREC_1(REQ := True,                                // Startimpuls
                ID := #hardwareId,                         // Diagnoseadresse
                INDEX := 47,                                  // Rahmentyp
                LEN := INT_TO_UINT(#piLenTele),             // maximale Länge
                DONE => #sbWrDone,                           // Schreibauftrag beendet
                BUSY => #sbWrBusy,                           // Slave beschäftigt
                ERROR => #sbWrError,                          // Fehler beim Schreiben
                STATUS => #pdStatus,                           // Status[1] = Error => Status[2] Error Decode + Status[3] Error Code
                RECORD := #sxChaParaMulti);                    // Zeiger auf zu schreibenen Datensatzes

       // Ausgänge setzen
       #sbBusy := #sbWrBusy;
       #sbDone := #sbWrDone;

       // Fehler auswerten
       IF #sbWrError THEN
         // Fehlerstatus aus dem Doppelwort filtern und weitergeben                
         #pwWord1 := DWORD_TO_WORD(SHR(IN := (#pdStatus AND DW#16#FFFF00), N := 8));

         // Fehlerstatus setzen
         #siErrorId := 3;
         #sbError := False;
         #DiagId := #pwWord1;

         //Temporärer Fehler: #pdStatus = 80A7, 80B5, 80C0, 80C1, 80C2, 80C3 oder 80C4 zulassen und nocheinmal versuchen
         IF NOT (#pwWord1 = DW#16#80A7) AND NOT (#pwWord1 = DW#16#80B5) AND NOT (#pwWord1 = DW#16#80C0) AND
           NOT (#pwWord1 = DW#16#80C1) AND NOT (#pwWord1 = DW#16#80C2) AND NOT (#pwWord1 = DW#16#80C3) AND
           NOT (#pwWord1 = DW#16#80C4) THEN

           // Wiederholungsauftrag wieder zurücknehmen
           #sbWrStart2 := False;
           #sbRdStart2 := False;
           #sbWrite := False;

           // Fehler ausgeben 
           #sbError := #sbWrError;

         ELSE
           // Fehlerwiederholauftrag ??                   
           IF #siErrorCount = #siMaxErrCount THEN

             // Wiederholungsauftrag wieder zurücknehmen
             #sbWrStart2 := False;
             #sbRdStart2 := False;
             #sbWrite := False;

             //Fehlerzähler zurücksetzen
             #siErrorCount := 0;


             // Fehler ausgeben 
             #sbError := #sbWrError;

             // nix tun bis Zähler überläuft
           ELSE
             #siErrorCount := #siErrorCount + 1;
           END_IF;
         END_IF;

         // kein Fehler beim SCHEIBEN AZYKLISCH und Auftrag fertig 
       ELSIF NOT #sbWrBusy AND #sbWrDone THEN
         // Fehlerkennung zurücknehmen
         #DiagId := W#16#00;

         // Schreibauftrag fertig melden und Leseantrag anstossen
         #sbWrStart2 := False;
         #sbRdStart2 := True;
       END_IF;
     END_IF; // 2. Teilauftrag "Parameter schreiben bzw. ändern" vorbereiten und abschicken

     // vom 2. Teilauftrag "Parameter schreiben bzw. ändern" die Antwort abwarten und dann auswerten
     IF #sbRdStart2 THEN

       // Ablöschen des Empfangspuffers
       #sxRespParaMulti.sxHeader.syReqRef := B#16#00;
       #sxRespParaMulti.sxHeader.syReqId := B#16#00;
       #sxRespParaMulti.sxHeader.syAxisNo := B#16#00;
       #sxRespParaMulti.sxHeader.syParaNo := B#16#00;

       FOR #piCount := 1 TO #siLenParaMulti DO
         #sxRespParaMulti.sxData[#piCount] := B#16#00;
       END_FOR;

       // LESEN AZYKLISCH
       #piLenTele := #siLenHeader + #siLenParaMulti;
       #RDREC_1(REQ := True,                                // Startimpuls
                ID := #hardwareId,                         // Diagnoseadresse        
                INDEX := 47,                                  // Rahmentyp           
                MLEN := INT_TO_UINT(#piLenTele),             // maximale Länge
                VALID => #pbValidSFB,                         // neuer Datensatz empfangen und gültig   
                BUSY => #sbRdBusy,                           // Slave beschäftigt
                ERROR => #sbRdError,                          // Fehler beim Schreiben
                STATUS => #pdStatus,                           // Status[1] = Error => Status[2] Error Decode + Status[3] Error Code 
                LEN => #piLenSFB,                           // Länge des gelesenen Datensatzes
                RECORD := #sxRespParaMulti);                   // Zeiger auf gelesenen Datensatz

       // Ausgänge setzen
       #sbBusy := #sbRdBusy;
       #sbDone := #pbValidSFB;

       // Fehler auswerten
       IF #sbRdError THEN
         // Fehlerstatus aus dem Doppelwort filtern und weitergeben                
         #pwWord1 := DWORD_TO_WORD(SHR(IN := (#pdStatus AND DW#16#FFFF00), N := 8));

         // Fehlerstatus setzen
         #siErrorId := 3;
         #DiagId := #pwWord1;

         //Temporärer Fehler: #pdStatus = 80A7, 80B5, 80C0, 80C1, 80C2, 80C3 oder 80C4 zulassen und nocheinmal versuchen
         IF NOT (#pwWord1 = DW#16#80A7) AND NOT (#pwWord1 = DW#16#80B5) AND NOT (#pwWord1 = DW#16#80C0) AND
           NOT (#pwWord1 = DW#16#80C1) AND NOT (#pwWord1 = DW#16#80C2) AND NOT (#pwWord1 = DW#16#80C3) AND
           NOT (#pwWord1 = DW#16#80C4) THEN

           // Wiederholungsauftrag wieder zurücknehmen
           #sbWrStart2 := False;
           #sbRdStart2 := False;
           #sbWrite := False;

           // Fehler ausgeben 
           #sbError := #sbRdError;

         ELSE
           // Fehlerwiederholauftrag ??                   
           IF #siErrorCount = #siMaxErrCount THEN

             // Wiederholungsauftrag wieder zurücknehmen
             #sbWrStart2 := False;
             #sbRdStart2 := False;
             #sbWrite := False;

             //Fehlerzähler zurücksetzen
             #siErrorCount := 0;


             // Fehler ausgeben 
             #sbError := #sbRdError;

             // nix tun bis Zähler überläuft
           ELSE
             #siErrorCount := #siErrorCount + 1;
           END_IF;
         END_IF;

         // Fehler : die Auftragsreferenz der Antwort übertimmt nicht mit der Auftragsreferenz der Anfrage überein
       ELSIF NOT (#siReqRef = BYTE_TO_INT(#sxRespParaMulti.sxHeader.syReqRef)) AND NOT #sbRdBusy AND #pbValidSFB THEN
         #siErrorId := 1;
         #sbError := True;
         #sbDone := False;

         // Wiederholungsauftrag wieder zurücknehmen
         #sbWrStart2 := False;
         #sbRdStart2 := False;
         #sbWrite := False;

         // Fehler : falsche Auftragskennung zurück erhalten    
       ELSIF NOT (#sxRespParaMulti.sxHeader.syReqId = B#16#82 OR #sxRespParaMulti.sxHeader.syReqId = B#16#02) AND
         NOT #sbRdBusy AND #pbValidSFB THEN
         #siErrorId := 1;
         #sbError := True;
         #sbDone := False;

         // Wiederholungsauftrag wieder zurücknehmen
         #sbWrStart2 := False;
         #sbRdStart2 := False;
         #sbWrite := False;

         // Fehler : die angeforderte Anzahl Parameter entspricht nicht der übermittelten Anzahl Parameter überein
       ELSIF NOT (#sxRespParaMulti.sxHeader.syParaNo = B#16#01) AND NOT #sbRdBusy AND #pbValidSFB THEN
         #siErrorId := 1;
         #sbError := True;
         #sbDone := False;

         // Wiederholungsauftrag wieder zurücknehmen
         #sbWrStart2 := False;
         #sbRdStart2 := False;
         #sbWrite := False;

         // Fehler : die Achse entspricht nicht der übergebenen Achse
       ELSIF NOT (#syAxisNo = #sxRespParaMulti.sxHeader.syAxisNo) AND NOT #sbRdBusy AND #pbValidSFB THEN
         #siErrorId := 1;
         #sbError := True;
         #sbDone := False;

         // Wiederholungsauftrag wieder zurücknehmen
         #sbWrStart2 := False;
         #sbRdStart2 := False;
         #sbWrite := False;

         // kein Fehler beim LESEN AZYKLISCH und Auftrag fertig 
       ELSIF NOT #sbRdBusy AND #pbValidSFB THEN

         // 2. Teilauftrag "Parameter schreiben bzw. ändern" negative Rückmeldung erhalten 
         IF #sxRespParaMulti.sxHeader.syReqId = B#16#82 THEN

           // die angefragten Parameter auswerten und im Puffer abspeichern
           // Format des Parameters auswerten, bei Format = Error Fehler auswerten 
           IF (BYTE_TO_INT(#sxRespParaMulti.sxData[1]) = 68) THEN

             // Fehlerwert ermitteln und abspeichern 
             // Format = Word, zwei Bytes zu übermitteltem Parameterwert zusammenfassen
             #pwWordHigh := SHL(IN := BYTE_TO_WORD(#sxRespParaMulti.sxData[3]), N := 8);
             #pwWordLow := BYTE_TO_WORD(#sxRespParaMulti.sxData[4]);
             #pwWord1 := #pwWordHigh XOR #pwWordLow;

             #sbError := True;

             // ermittelte Fehlernummer im Puffer zurücksetzen
             #ErrorNo := W#16#00;

             #ErrorNo := #pwWord1;

             // Die Fehlerhaftigkeit des erkannten Parameter in der Fehlernummer eintragen   
             #swParaError := #swParaError OR W#16#01;

           ELSE

             // Die Fehlerhaftigkeit des erkannten Parameter in der Fehlernummer löschen   
             #swParaError := #swParaError AND W#16#FFFE;

             // ermittelte Fehlernummer im Puffer zurücksetzen
             #ErrorNo := W#16#00;
           END_IF;
         END_IF; // 2. Teilauftrag "Parameter schreiben bzw. ändern" negative Rückmeldung erhalten

         // Fehlerkennung zurücknehmen
         IF (#siErrorId = 3) OR (#siErrorId = 1) THEN
           #siErrorId := 0;
           #sbError := False;
         END_IF;

         #DiagId := W#16#00;

         // 2. Teilauftrag "Parameter schreiben bzw. ändern" ist abgeschlossen
         #sbRdStart2 := False;
         #sbWrite := False;

       END_IF; // kein Fehler beim LESEN AZYKLISCH und Auftrag fertig 
     END_IF; // vom 2. Teilauftrag "Parameter schreiben bzw. ändern" die Antwort abwarten und dann auswerten 
   END_IF; // Auftrag "Parameter schreiben" wurde ausgelöst

   #pdDWordHigh := SHL(IN := INT_TO_DWORD(#siErrorId), N := 16);
   #pdDWordLow := WORD_TO_DWORD(#swParaError);

   // ermittelter Parameterwert eintragen (Word)
   #ErrorId := #pdDWordHigh XOR #pdDWordLow;

   // Initialisierung von Ausgängen
   #Busy := #sbBusy;
   #Error := #sbError;
   #Format := #syFormat;
   // Änderung wegen verhalten von Ready  
   #Done := #sbDone;
   // Prüfen, ob Auftrag abgeschlossen ist
   IF ((#Error OR #Done) AND NOT #sbReady) THEN
     #Ready := True;
     #sbReady := True;
   ELSE
     #Ready := False;
   END_IF;
END_FUNCTION_BLOCK

DATA_BLOCK "ST10_FB_Tower_4Lamp_DB"   // DB5050
// stored: AutoNumber false, InstanceOfName FB_Tower_4Lamp, InstanceOfType FB
"FB_Tower_4Lamp"
BEGIN
END_DATA_BLOCK

DATA_BLOCK "ST10_CountCycleTimeMain_DB"   // DB1009
// stored: AutoNumber false, InstanceOfName ST10_CountCycleTimeMain, InstanceOfType FB
"ST10_CountCycleTimeMain"
BEGIN
END_DATA_BLOCK

DATA_BLOCK "DT-Chars_DB"   // DB2360
// stored: AutoNumber false, InstanceOfName DT-Chars, InstanceOfType FB
"DT-Chars"
BEGIN
END_DATA_BLOCK

DATA_BLOCK "FB_MES_Monitoring_iDB"   // DB10
// stored: InstanceOfName FB_MES_Monitoring, InstanceOfType FB
"FB_MES_Monitoring"
BEGIN
END_DATA_BLOCK

DATA_BLOCK "MES_CHeck_DB"   // DB111
// stored: AutoNumber false, InstanceOfName MES_CHeck, InstanceOfType FB
"MES_CHeck"
BEGIN
END_DATA_BLOCK

DATA_BLOCK "PartDataManage_Part1_DB"   // DB1501
// stored: InstanceOfName PartDataManage, InstanceOfType FB
"PartDataManage"
BEGIN
END_DATA_BLOCK

DATA_BLOCK "PartDataManage_Part2_DB"   // DB1502
// stored: InstanceOfName PartDataManage, InstanceOfType FB
"PartDataManage"
BEGIN
END_DATA_BLOCK

DATA_BLOCK "PartDataManage_Part3_DB"   // DB1503
// stored: InstanceOfName PartDataManage, InstanceOfType FB
"PartDataManage"
BEGIN
END_DATA_BLOCK

DATA_BLOCK "PartDataManage_Part4_DB"   // DB1504
// stored: InstanceOfName PartDataManage, InstanceOfType FB
"PartDataManage"
BEGIN
END_DATA_BLOCK

DATA_BLOCK "ST10_SystemModeFB_iDB"   // DB1000
// stored: AutoNumber false, InstanceOfName SystemMode, InstanceOfType FB
"SystemMode"
BEGIN
END_DATA_BLOCK

DATA_BLOCK "ST10_Flow5_FRobot_1_DB"   // DB13
// stored: AutoNumber false, InstanceOfName ST10_Flow5_FRobot_1, InstanceOfType FB
"ST10_Flow5_FRobot_1"
BEGIN
END_DATA_BLOCK

DATA_BLOCK "AutoProcessDataPopUp_DB"   // DB2
// stored: InstanceOfName AutoProcessDataPopUp, InstanceOfType FB
"AutoProcessDataPopUp"
BEGIN
END_DATA_BLOCK

DATA_BLOCK "ST10_Flow11_A2TableScan_iDB"   // DB1081
// stored: AutoNumber false, InstanceOfName ST10_Flow11_A2TableScan, InstanceOfType FB
"ST10_Flow11_A2TableScan"
BEGIN
END_DATA_BLOCK

DATA_BLOCK "ST10_Flow12_A2TableUnloading_iDB"   // DB1082
// stored: AutoNumber false, InstanceOfName ST10_Flow12_A2TableUnloading, InstanceOfType FB
"ST10_Flow12_A2TableUnloading"
BEGIN
END_DATA_BLOCK

DATA_BLOCK "ST10_Flow14_B2Press_iDB"   // DB1084
// stored: AutoNumber false, InstanceOfName ST10_Flow14_B2Press, InstanceOfType FB
"ST10_Flow14_B2Press"
BEGIN
END_DATA_BLOCK

DATA_BLOCK "ST10_Flow15_FRobot_3_iDB"   // DB1085
// stored: AutoNumber false, InstanceOfName ST10_Flow15_FRobot_3, InstanceOfType FB
"ST10_Flow15_FRobot_3"
BEGIN
END_DATA_BLOCK

DATA_BLOCK "ST10_Flow1_A1TableScan_iDB"   // DB1071
// stored: AutoNumber false, InstanceOfName ST10_Flow1_A1TableScan, InstanceOfType FB
"ST10_Flow1_A1TableScan"
BEGIN
END_DATA_BLOCK

DATA_BLOCK "ST10_Flow21_HShaftLifting_iDB"   // DB1091
// stored: AutoNumber false, InstanceOfName ST10_Flow21_HShaftLifting, InstanceOfType FB
"ST10_Flow21_HShaftLifting"
BEGIN
END_DATA_BLOCK

DATA_BLOCK "ST10_Flow22_JMagnetLifting_iDB"   // DB1092
// stored: AutoNumber false, InstanceOfName ST10_Flow22_JMagnetLifting, InstanceOfType FB
"ST10_Flow22_JMagnetLifting"
BEGIN
END_DATA_BLOCK

DATA_BLOCK "ST10_Flow23_KReserveLifting_iDB"   // DB1093
// stored: AutoNumber false, InstanceOfName ST10_Flow23_KReserveLifting, InstanceOfType FB
"ST10_Flow23_KReserveLifting"
BEGIN
END_DATA_BLOCK

DATA_BLOCK "ST10_Flow24_LUnloadingTrans_iDB"   // DB1094
// stored: AutoNumber false, InstanceOfName ST10_Flow24_LUnloadingTrans, InstanceOfType FB
"ST10_Flow24_LUnloadingTrans"
BEGIN
END_DATA_BLOCK

DATA_BLOCK "ST10_Flow25_HShaftLoad&Unload_iDB"   // DB1095
// stored: AutoNumber false, InstanceOfName ST10_Flow25_HShaftLoad&Unload, InstanceOfType FB
"ST10_Flow25_HShaftLoad&Unload"
BEGIN
END_DATA_BLOCK

DATA_BLOCK "ST10_Flow26_JMagnetLoad&Unload_iDB"   // DB1096
// stored: AutoNumber false, InstanceOfName ST10_Flow26_JMagnetLoad&Unload, InstanceOfType FB
"ST10_Flow26_JMagnetLoad&Unload"
BEGIN
END_DATA_BLOCK

